// TwinCAT 3 PLC project PLC
// ProgramVersion: 3.1.4023.0
// libraries:
//   Tc2_Standard, * (Beckhoff Automation GmbH)
//   Tc2_System, * (Beckhoff Automation GmbH)
//   Tc3_Module, * (Beckhoff Automation GmbH)
// project tree:
//   / PlcTask.TcTTO
//   POUs/ MAIN.TcPOU
//   DUTs/IO/PdoEntries/ Status_B0753356.TcDUT, Status_F2CE6D91.TcDUT
//   DUTs/IO/PDOs/ InfoData_6F19DB2B.TcDUT, Channel_830843C1.TcDUT, WcState_9091E0EB.TcDUT, Channel_42CA91F7.TcDUT, WcState_0B2B16F9.TcDUT, AI_Standard_Channel_A8DF64E3.TcDUT, InfoData_32EB74EA.TcDUT, RTD_RTDInputs_Channel_A8DF64E3.TcDUT, AI_Standard_Channel_4A394481.TcDUT, TC_TCInputs_Channel_A8DF64E3.TcDUT, InfoData_E68C61CD.TcDUT, InfoData_2A97D6CF.TcDUT, Inputs_25A0042B.TcDUT, Outputs_2397A10E.TcDUT
//   DUTs/IO/Boxes/ EK1100_1FC0878B.TcDUT, EK1122_1FC0878B.TcDUT, EQ1008_78E8D3DD.TcDUT, EQ1809_32157CFD.TcDUT, EQ2008_E2806B95.TcDUT, EQ2339_4CF33DED.TcDUT, EQ2809_2B6483BD.TcDUT, EQ3174_DCC78662.TcDUT, EQ3204_6CD7E119.TcDUT, EQ3204_AB25C3AC.TcDUT, EQ3314_1CEB931C.TcDUT, EQ3314_E65CDB1C.TcDUT
//   DUTs/IO/Devices/ SyncUnitTask_2D604ED5.TcDUT, SyncUnitTasks_6FEB8257.TcDUT, SyncUnits_99E584AF.TcDUT
//   DUTs/IO/Topology/ Beckhoff_EQ1xxxEK1122_E78E0C94.TcDUT, Beckhoff_EQ1xxx_F67C323D.TcDUT, Beckhoff_EQ2xxxEK1122_214B8BB9.TcDUT, Beckhoff_EQ2xxx_A19B669C.TcDUT, Beckhoff_EQ3xxxEK1122_A1C56A21.TcDUT, Beckhoff_EQ3xxx_A920B096.TcDUT, EtherCAT_Master_EQxxxx_806C2CF0.TcDUT
//   DUTs/IO/Base/ EtcSlaveBase_82538BE2.TcDUT, EtcSlaveBase_82538BE2.TcDUT, EtcSlaveBase_82538BE2.TcDUT, EtcSlaveTerminalBase_947E5A46.TcDUT, EtcSlaveBoxBase_77A0E4A7.TcDUT, EtcSlaveEndTerminalBase_866C7F0C.TcDUT, InputBase_8311D824.TcDUT, OutputBase_10CEE7DE.TcDUT, EtcMasterBase_62654B43.TcDUT
//   GVLs/ GVL_iXlinker.TcGVL
// real-time tasks:
//   TASK PlcTask: cycle T#10ms, priority 20, ADS port 350
// I/O:
//   DEVICE EtherCAT_Master_EQxxxx, AmsNetId 172.20.30.238.15.1
//     Beckhoff EQ1xxx [EK1100 EtherCAT Coupler (2A E-Bus)]
//       Beckhoff EQ1xxxEK1122 [EK1122 2 port EtherCAT junction]
//         Beckhoff EQ1xxxsub EK1100 [EK1100 EtherCAT Coupler (2A E-Bus)]
//         A_0001(EQ1008-0002-0016) [EQ1008-0002 8 Ch. Dig. Input 24V, 3ms, M12]
//         A_0002(EQ1008-0002-0017) [EQ1008-0002 8 Ch. Dig. Input 24V, 3ms, M12]
//         A_0003(EQ1008-0002-0018) [EQ1008-0002 8 Ch. Dig. Input 24V, 3ms, M12]
//         A_0004(EQ1809-0022-0016) [EQ1809-0022 16 Ch. Dig. Input 24V, 3ms, M12]
//         A_0005(EQ1809-0022-0018) [EQ1809-0022 16 Ch. Dig. Input 24V, 3ms, M12]
//     Beckhoff EQ2xxx [EK1100 EtherCAT Coupler (2A E-Bus)]
//       Beckhoff EQ2xxxEK1122 [EK1122 2 port EtherCAT junction]
//         Beckhoff EQ2xxxsub EK1100 [EK1100 EtherCAT Coupler (2A E-Bus)]
//         A_0001(EQ2008-0002-0016) [EQ2008-0002 8 Ch. Dig. Output 24V, 0,5A, M12]
//         A_0002(EQ2008-0002-0017) [EQ2008-0002 8 Ch. Dig. Output 24V, 0,5A, M12]
//         A_0003(EQ2008-0002-0018) [EQ2008-0002 8 Ch. Dig. Output 24V, 0,5A, M12]
//         A_0004(EQ2008-0002-0019) [EQ2008-0002 8 Ch. Dig. Output 24V, 0,5A, M12]
//         A_0005(EQ2339-0022-0016) [EQ2339-0022 16 Ch. Dig. Input/Output 24V, 0,5A, M12]
//         A_0006(EQ2339-0022-0017) [EQ2339-0022 16 Ch. Dig. Input/Output 24V, 0,5A, M12]
//         A_0007(EQ2339-0022-0018) [EQ2339-0022 16 Ch. Dig. Input/Output 24V, 0,5A, M12]
//         A_0008(EQ2339-0022-0019) [EQ2339-0022 16 Ch. Dig. Input/Output 24V, 0,5A, M12]
//         A_0009(EQ2809-0022-0016) [EQ2809-0022 16 Ch. Dig. Output 24V, 0,5A, M12]
//         A_0010(EQ2809-0022-0017) [EQ2809-0022 16 Ch. Dig. Output 24V, 0,5A, M12]
//         A_0011(EQ2809-0022-0018) [EQ2809-0022 16 Ch. Dig. Output 24V, 0,5A, M12]
//     Beckhoff EQ3xxx [EK1100 EtherCAT Coupler (2A E-Bus)]
//       Beckhoff EQ3xxxEK1122 [EK1122 2 port EtherCAT junction]
//         Beckhoff EQ3xxxsub EK1100 [EK1100 EtherCAT Coupler (2A E-Bus)]
//         A_0001(EQ3174-0002-0016) [EQ3174-0002 4Ch. Ana. Input +/-10V, 0-10V, 0/4-20mA configurable]
//         A_0002(EQ3174-0002-0017) [EQ3174-0002 4Ch. Ana. Input +/-10V, 0-10V, 0/4-20mA configurable]
//         A_0003(EQ3174-0002-0021) [EQ3174-0002 4Ch. Ana. Input +/-10V, 0-10V, 0/4-20mA configurable]
//         A_0004(EQ3174-0002-0022) [EQ3174-0002 4Ch. Ana. Input +/-10V, 0-10V, 0/4-20mA configurable]
//         A_0005(EQ3174-0002-0023) [EQ3174-0002 4Ch. Ana. Input +/-10V, 0-10V, 0/4-20mA configurable]
//         A_0006(EQ3204-0002-0016) [EQ3204-0002 4Ch. Ana. Input PT100 (RTD)]
//         A_0007(EQ3204-0002-0017) [EQ3204-0002 4Ch. Ana. Input PT100 (RTD)]
//         A_0008(EQ3204-0002-0020) [EQ3204-0002 4Ch. Ana. Input PT100 (RTD)]
//         A_0009(EQ3204-0002-0021) [EQ3204-0002 4Ch. Ana. Input PT100 (RTD)]
//         A_0010(EQ3204-0002-0022) [EQ3204-0002 4Ch. Ana. Input PT100 (RTD)]
//         A_0011(EQ3314-0002-0016) [EQ3314-0002 4Ch. Ana. Input Thermocouple (TC)]
//         A_0012(EQ3314-0002-0017) [EQ3314-0002 4Ch. Ana. Input Thermocouple (TC)]
//         A_0013(EQ3314-0002-0021) [EQ3314-0002 4Ch. Ana. Input Thermocouple (TC)]
//         A_0014(EQ3314-0002-0022) [EQ3314-0002 4Ch. Ana. Input Thermocouple (TC)]
// variable links:
//   PLC/PLC Instance <-> EtherCAT Master EQxxxx/Beckhoff EQ1xxx
//     PlcTask Inputs/GVL_iXlinker.EtherCAT_Master_EQxxxx.Beckhoff_EQ1xxx.InfoData.State <-> InfoData/State
//   PLC/PLC Instance <-> EtherCAT Master EQxxxx/Beckhoff EQ1xxx/Beckhoff EQ1xxxEK1122
//     PlcTask Inputs/GVL_iXlinker.EtherCAT_Master_EQxxxx.Beckhoff_EQ1xxx.Beckhoff_EQ1xxxEK1122.InfoData.State <-> InfoData/State
//   PLC/PLC Instance <-> EtherCAT Master EQxxxx/Beckhoff EQ1xxx/Beckhoff EQ1xxxEK1122/Beckhoff EQ1xxxsub EK1100
//     PlcTask Inputs/GVL_iXlinker.EtherCAT_Master_EQxxxx.Beckhoff_EQ1xxx.Beckhoff_EQ1xxxEK1122.Beckhoff_EQ1xxxsub_EK1100.InfoData.State <-> InfoData/State
//   PLC/PLC Instance <-> EtherCAT Master EQxxxx/Beckhoff EQ1xxx/Beckhoff EQ1xxxEK1122/A_0001(EQ1008-0002-0016)
//     PlcTask Inputs/GVL_iXlinker.EtherCAT_Master_EQxxxx.Beckhoff_EQ1xxx.Beckhoff_EQ1xxxEK1122.A_0001_EQ1008_0002_0016.Channel_1.Input <-> Channel 1/Input
//     PlcTask Inputs/GVL_iXlinker.EtherCAT_Master_EQxxxx.Beckhoff_EQ1xxx.Beckhoff_EQ1xxxEK1122.A_0001_EQ1008_0002_0016.Channel_2.Input <-> Channel 2/Input
//     PlcTask Inputs/GVL_iXlinker.EtherCAT_Master_EQxxxx.Beckhoff_EQ1xxx.Beckhoff_EQ1xxxEK1122.A_0001_EQ1008_0002_0016.Channel_3.Input <-> Channel 3/Input
//     PlcTask Inputs/GVL_iXlinker.EtherCAT_Master_EQxxxx.Beckhoff_EQ1xxx.Beckhoff_EQ1xxxEK1122.A_0001_EQ1008_0002_0016.Channel_4.Input <-> Channel 4/Input
//     PlcTask Inputs/GVL_iXlinker.EtherCAT_Master_EQxxxx.Beckhoff_EQ1xxx.Beckhoff_EQ1xxxEK1122.A_0001_EQ1008_0002_0016.Channel_5.Input <-> Channel 5/Input
//     PlcTask Inputs/GVL_iXlinker.EtherCAT_Master_EQxxxx.Beckhoff_EQ1xxx.Beckhoff_EQ1xxxEK1122.A_0001_EQ1008_0002_0016.Channel_6.Input <-> Channel 6/Input
//     PlcTask Inputs/GVL_iXlinker.EtherCAT_Master_EQxxxx.Beckhoff_EQ1xxx.Beckhoff_EQ1xxxEK1122.A_0001_EQ1008_0002_0016.Channel_7.Input <-> Channel 7/Input
//     PlcTask Inputs/GVL_iXlinker.EtherCAT_Master_EQxxxx.Beckhoff_EQ1xxx.Beckhoff_EQ1xxxEK1122.A_0001_EQ1008_0002_0016.Channel_8.Input <-> Channel 8/Input
//     PlcTask Inputs/GVL_iXlinker.EtherCAT_Master_EQxxxx.Beckhoff_EQ1xxx.Beckhoff_EQ1xxxEK1122.A_0001_EQ1008_0002_0016.WcState.WcState <-> WcState/WcState
//     PlcTask Inputs/GVL_iXlinker.EtherCAT_Master_EQxxxx.Beckhoff_EQ1xxx.Beckhoff_EQ1xxxEK1122.A_0001_EQ1008_0002_0016.WcState.InputToggle <-> WcState/InputToggle
//     PlcTask Inputs/GVL_iXlinker.EtherCAT_Master_EQxxxx.Beckhoff_EQ1xxx.Beckhoff_EQ1xxxEK1122.A_0001_EQ1008_0002_0016.InfoData.State <-> InfoData/State
//   PLC/PLC Instance <-> EtherCAT Master EQxxxx/Beckhoff EQ1xxx/Beckhoff EQ1xxxEK1122/A_0002(EQ1008-0002-0017)
//     PlcTask Inputs/GVL_iXlinker.EtherCAT_Master_EQxxxx.Beckhoff_EQ1xxx.Beckhoff_EQ1xxxEK1122.A_0002_EQ1008_0002_0017.Channel_1.Input <-> Channel 1/Input
//     PlcTask Inputs/GVL_iXlinker.EtherCAT_Master_EQxxxx.Beckhoff_EQ1xxx.Beckhoff_EQ1xxxEK1122.A_0002_EQ1008_0002_0017.Channel_2.Input <-> Channel 2/Input
//     PlcTask Inputs/GVL_iXlinker.EtherCAT_Master_EQxxxx.Beckhoff_EQ1xxx.Beckhoff_EQ1xxxEK1122.A_0002_EQ1008_0002_0017.Channel_3.Input <-> Channel 3/Input
//     PlcTask Inputs/GVL_iXlinker.EtherCAT_Master_EQxxxx.Beckhoff_EQ1xxx.Beckhoff_EQ1xxxEK1122.A_0002_EQ1008_0002_0017.Channel_4.Input <-> Channel 4/Input
//     PlcTask Inputs/GVL_iXlinker.EtherCAT_Master_EQxxxx.Beckhoff_EQ1xxx.Beckhoff_EQ1xxxEK1122.A_0002_EQ1008_0002_0017.Channel_5.Input <-> Channel 5/Input
//     PlcTask Inputs/GVL_iXlinker.EtherCAT_Master_EQxxxx.Beckhoff_EQ1xxx.Beckhoff_EQ1xxxEK1122.A_0002_EQ1008_0002_0017.Channel_6.Input <-> Channel 6/Input
//     PlcTask Inputs/GVL_iXlinker.EtherCAT_Master_EQxxxx.Beckhoff_EQ1xxx.Beckhoff_EQ1xxxEK1122.A_0002_EQ1008_0002_0017.Channel_7.Input <-> Channel 7/Input
//     PlcTask Inputs/GVL_iXlinker.EtherCAT_Master_EQxxxx.Beckhoff_EQ1xxx.Beckhoff_EQ1xxxEK1122.A_0002_EQ1008_0002_0017.Channel_8.Input <-> Channel 8/Input
//     PlcTask Inputs/GVL_iXlinker.EtherCAT_Master_EQxxxx.Beckhoff_EQ1xxx.Beckhoff_EQ1xxxEK1122.A_0002_EQ1008_0002_0017.WcState.WcState <-> WcState/WcState
//     PlcTask Inputs/GVL_iXlinker.EtherCAT_Master_EQxxxx.Beckhoff_EQ1xxx.Beckhoff_EQ1xxxEK1122.A_0002_EQ1008_0002_0017.WcState.InputToggle <-> WcState/InputToggle
//     PlcTask Inputs/GVL_iXlinker.EtherCAT_Master_EQxxxx.Beckhoff_EQ1xxx.Beckhoff_EQ1xxxEK1122.A_0002_EQ1008_0002_0017.InfoData.State <-> InfoData/State
//   PLC/PLC Instance <-> EtherCAT Master EQxxxx/Beckhoff EQ1xxx/Beckhoff EQ1xxxEK1122/A_0003(EQ1008-0002-0018)
//     PlcTask Inputs/GVL_iXlinker.EtherCAT_Master_EQxxxx.Beckhoff_EQ1xxx.Beckhoff_EQ1xxxEK1122.A_0003_EQ1008_0002_0018.Channel_1.Input <-> Channel 1/Input
//     PlcTask Inputs/GVL_iXlinker.EtherCAT_Master_EQxxxx.Beckhoff_EQ1xxx.Beckhoff_EQ1xxxEK1122.A_0003_EQ1008_0002_0018.Channel_2.Input <-> Channel 2/Input
//     PlcTask Inputs/GVL_iXlinker.EtherCAT_Master_EQxxxx.Beckhoff_EQ1xxx.Beckhoff_EQ1xxxEK1122.A_0003_EQ1008_0002_0018.Channel_3.Input <-> Channel 3/Input
//     PlcTask Inputs/GVL_iXlinker.EtherCAT_Master_EQxxxx.Beckhoff_EQ1xxx.Beckhoff_EQ1xxxEK1122.A_0003_EQ1008_0002_0018.Channel_4.Input <-> Channel 4/Input
//     PlcTask Inputs/GVL_iXlinker.EtherCAT_Master_EQxxxx.Beckhoff_EQ1xxx.Beckhoff_EQ1xxxEK1122.A_0003_EQ1008_0002_0018.Channel_5.Input <-> Channel 5/Input
//     PlcTask Inputs/GVL_iXlinker.EtherCAT_Master_EQxxxx.Beckhoff_EQ1xxx.Beckhoff_EQ1xxxEK1122.A_0003_EQ1008_0002_0018.Channel_6.Input <-> Channel 6/Input
//     PlcTask Inputs/GVL_iXlinker.EtherCAT_Master_EQxxxx.Beckhoff_EQ1xxx.Beckhoff_EQ1xxxEK1122.A_0003_EQ1008_0002_0018.Channel_7.Input <-> Channel 7/Input
//     PlcTask Inputs/GVL_iXlinker.EtherCAT_Master_EQxxxx.Beckhoff_EQ1xxx.Beckhoff_EQ1xxxEK1122.A_0003_EQ1008_0002_0018.Channel_8.Input <-> Channel 8/Input
//     PlcTask Inputs/GVL_iXlinker.EtherCAT_Master_EQxxxx.Beckhoff_EQ1xxx.Beckhoff_EQ1xxxEK1122.A_0003_EQ1008_0002_0018.WcState.WcState <-> WcState/WcState
//     PlcTask Inputs/GVL_iXlinker.EtherCAT_Master_EQxxxx.Beckhoff_EQ1xxx.Beckhoff_EQ1xxxEK1122.A_0003_EQ1008_0002_0018.WcState.InputToggle <-> WcState/InputToggle
//     PlcTask Inputs/GVL_iXlinker.EtherCAT_Master_EQxxxx.Beckhoff_EQ1xxx.Beckhoff_EQ1xxxEK1122.A_0003_EQ1008_0002_0018.InfoData.State <-> InfoData/State
//   PLC/PLC Instance <-> EtherCAT Master EQxxxx/Beckhoff EQ1xxx/Beckhoff EQ1xxxEK1122/A_0004(EQ1809-0022-0016)
//     PlcTask Inputs/GVL_iXlinker.EtherCAT_Master_EQxxxx.Beckhoff_EQ1xxx.Beckhoff_EQ1xxxEK1122.A_0004_EQ1809_0022_0016.Channel_1.Input <-> Channel 1/Input
//     PlcTask Inputs/GVL_iXlinker.EtherCAT_Master_EQxxxx.Beckhoff_EQ1xxx.Beckhoff_EQ1xxxEK1122.A_0004_EQ1809_0022_0016.Channel_2.Input <-> Channel 2/Input
//     PlcTask Inputs/GVL_iXlinker.EtherCAT_Master_EQxxxx.Beckhoff_EQ1xxx.Beckhoff_EQ1xxxEK1122.A_0004_EQ1809_0022_0016.Channel_3.Input <-> Channel 3/Input
//     PlcTask Inputs/GVL_iXlinker.EtherCAT_Master_EQxxxx.Beckhoff_EQ1xxx.Beckhoff_EQ1xxxEK1122.A_0004_EQ1809_0022_0016.Channel_4.Input <-> Channel 4/Input
//     PlcTask Inputs/GVL_iXlinker.EtherCAT_Master_EQxxxx.Beckhoff_EQ1xxx.Beckhoff_EQ1xxxEK1122.A_0004_EQ1809_0022_0016.Channel_5.Input <-> Channel 5/Input
//     PlcTask Inputs/GVL_iXlinker.EtherCAT_Master_EQxxxx.Beckhoff_EQ1xxx.Beckhoff_EQ1xxxEK1122.A_0004_EQ1809_0022_0016.Channel_6.Input <-> Channel 6/Input
//     PlcTask Inputs/GVL_iXlinker.EtherCAT_Master_EQxxxx.Beckhoff_EQ1xxx.Beckhoff_EQ1xxxEK1122.A_0004_EQ1809_0022_0016.Channel_7.Input <-> Channel 7/Input
//     PlcTask Inputs/GVL_iXlinker.EtherCAT_Master_EQxxxx.Beckhoff_EQ1xxx.Beckhoff_EQ1xxxEK1122.A_0004_EQ1809_0022_0016.Channel_8.Input <-> Channel 8/Input
//     PlcTask Inputs/GVL_iXlinker.EtherCAT_Master_EQxxxx.Beckhoff_EQ1xxx.Beckhoff_EQ1xxxEK1122.A_0004_EQ1809_0022_0016.Channel_9.Input <-> Channel 9/Input
//     PlcTask Inputs/GVL_iXlinker.EtherCAT_Master_EQxxxx.Beckhoff_EQ1xxx.Beckhoff_EQ1xxxEK1122.A_0004_EQ1809_0022_0016.Channel_10.Input <-> Channel 10/Input
//     PlcTask Inputs/GVL_iXlinker.EtherCAT_Master_EQxxxx.Beckhoff_EQ1xxx.Beckhoff_EQ1xxxEK1122.A_0004_EQ1809_0022_0016.Channel_11.Input <-> Channel 11/Input
//     PlcTask Inputs/GVL_iXlinker.EtherCAT_Master_EQxxxx.Beckhoff_EQ1xxx.Beckhoff_EQ1xxxEK1122.A_0004_EQ1809_0022_0016.Channel_12.Input <-> Channel 12/Input
//     PlcTask Inputs/GVL_iXlinker.EtherCAT_Master_EQxxxx.Beckhoff_EQ1xxx.Beckhoff_EQ1xxxEK1122.A_0004_EQ1809_0022_0016.Channel_13.Input <-> Channel 13/Input
//     PlcTask Inputs/GVL_iXlinker.EtherCAT_Master_EQxxxx.Beckhoff_EQ1xxx.Beckhoff_EQ1xxxEK1122.A_0004_EQ1809_0022_0016.Channel_14.Input <-> Channel 14/Input
//     PlcTask Inputs/GVL_iXlinker.EtherCAT_Master_EQxxxx.Beckhoff_EQ1xxx.Beckhoff_EQ1xxxEK1122.A_0004_EQ1809_0022_0016.Channel_15.Input <-> Channel 15/Input
//     PlcTask Inputs/GVL_iXlinker.EtherCAT_Master_EQxxxx.Beckhoff_EQ1xxx.Beckhoff_EQ1xxxEK1122.A_0004_EQ1809_0022_0016.Channel_16.Input <-> Channel 16/Input
//     PlcTask Inputs/GVL_iXlinker.EtherCAT_Master_EQxxxx.Beckhoff_EQ1xxx.Beckhoff_EQ1xxxEK1122.A_0004_EQ1809_0022_0016.WcState.WcState <-> WcState/WcState
//     PlcTask Inputs/GVL_iXlinker.EtherCAT_Master_EQxxxx.Beckhoff_EQ1xxx.Beckhoff_EQ1xxxEK1122.A_0004_EQ1809_0022_0016.WcState.InputToggle <-> WcState/InputToggle
//     PlcTask Inputs/GVL_iXlinker.EtherCAT_Master_EQxxxx.Beckhoff_EQ1xxx.Beckhoff_EQ1xxxEK1122.A_0004_EQ1809_0022_0016.InfoData.State <-> InfoData/State
//   PLC/PLC Instance <-> EtherCAT Master EQxxxx/Beckhoff EQ1xxx/Beckhoff EQ1xxxEK1122/A_0005(EQ1809-0022-0018)
//     PlcTask Inputs/GVL_iXlinker.EtherCAT_Master_EQxxxx.Beckhoff_EQ1xxx.Beckhoff_EQ1xxxEK1122.A_0005_EQ1809_0022_0018.Channel_1.Input <-> Channel 1/Input
//     PlcTask Inputs/GVL_iXlinker.EtherCAT_Master_EQxxxx.Beckhoff_EQ1xxx.Beckhoff_EQ1xxxEK1122.A_0005_EQ1809_0022_0018.Channel_2.Input <-> Channel 2/Input
//     PlcTask Inputs/GVL_iXlinker.EtherCAT_Master_EQxxxx.Beckhoff_EQ1xxx.Beckhoff_EQ1xxxEK1122.A_0005_EQ1809_0022_0018.Channel_3.Input <-> Channel 3/Input
//     PlcTask Inputs/GVL_iXlinker.EtherCAT_Master_EQxxxx.Beckhoff_EQ1xxx.Beckhoff_EQ1xxxEK1122.A_0005_EQ1809_0022_0018.Channel_4.Input <-> Channel 4/Input
//     PlcTask Inputs/GVL_iXlinker.EtherCAT_Master_EQxxxx.Beckhoff_EQ1xxx.Beckhoff_EQ1xxxEK1122.A_0005_EQ1809_0022_0018.Channel_5.Input <-> Channel 5/Input
//     PlcTask Inputs/GVL_iXlinker.EtherCAT_Master_EQxxxx.Beckhoff_EQ1xxx.Beckhoff_EQ1xxxEK1122.A_0005_EQ1809_0022_0018.Channel_6.Input <-> Channel 6/Input
//     PlcTask Inputs/GVL_iXlinker.EtherCAT_Master_EQxxxx.Beckhoff_EQ1xxx.Beckhoff_EQ1xxxEK1122.A_0005_EQ1809_0022_0018.Channel_7.Input <-> Channel 7/Input
//     PlcTask Inputs/GVL_iXlinker.EtherCAT_Master_EQxxxx.Beckhoff_EQ1xxx.Beckhoff_EQ1xxxEK1122.A_0005_EQ1809_0022_0018.Channel_8.Input <-> Channel 8/Input
//     PlcTask Inputs/GVL_iXlinker.EtherCAT_Master_EQxxxx.Beckhoff_EQ1xxx.Beckhoff_EQ1xxxEK1122.A_0005_EQ1809_0022_0018.Channel_9.Input <-> Channel 9/Input
//     PlcTask Inputs/GVL_iXlinker.EtherCAT_Master_EQxxxx.Beckhoff_EQ1xxx.Beckhoff_EQ1xxxEK1122.A_0005_EQ1809_0022_0018.Channel_10.Input <-> Channel 10/Input
//     PlcTask Inputs/GVL_iXlinker.EtherCAT_Master_EQxxxx.Beckhoff_EQ1xxx.Beckhoff_EQ1xxxEK1122.A_0005_EQ1809_0022_0018.Channel_11.Input <-> Channel 11/Input
//     PlcTask Inputs/GVL_iXlinker.EtherCAT_Master_EQxxxx.Beckhoff_EQ1xxx.Beckhoff_EQ1xxxEK1122.A_0005_EQ1809_0022_0018.Channel_12.Input <-> Channel 12/Input
//     PlcTask Inputs/GVL_iXlinker.EtherCAT_Master_EQxxxx.Beckhoff_EQ1xxx.Beckhoff_EQ1xxxEK1122.A_0005_EQ1809_0022_0018.Channel_13.Input <-> Channel 13/Input
//     PlcTask Inputs/GVL_iXlinker.EtherCAT_Master_EQxxxx.Beckhoff_EQ1xxx.Beckhoff_EQ1xxxEK1122.A_0005_EQ1809_0022_0018.Channel_14.Input <-> Channel 14/Input
//     PlcTask Inputs/GVL_iXlinker.EtherCAT_Master_EQxxxx.Beckhoff_EQ1xxx.Beckhoff_EQ1xxxEK1122.A_0005_EQ1809_0022_0018.Channel_15.Input <-> Channel 15/Input
//     PlcTask Inputs/GVL_iXlinker.EtherCAT_Master_EQxxxx.Beckhoff_EQ1xxx.Beckhoff_EQ1xxxEK1122.A_0005_EQ1809_0022_0018.Channel_16.Input <-> Channel 16/Input
//     PlcTask Inputs/GVL_iXlinker.EtherCAT_Master_EQxxxx.Beckhoff_EQ1xxx.Beckhoff_EQ1xxxEK1122.A_0005_EQ1809_0022_0018.WcState.WcState <-> WcState/WcState
//     PlcTask Inputs/GVL_iXlinker.EtherCAT_Master_EQxxxx.Beckhoff_EQ1xxx.Beckhoff_EQ1xxxEK1122.A_0005_EQ1809_0022_0018.WcState.InputToggle <-> WcState/InputToggle
//     PlcTask Inputs/GVL_iXlinker.EtherCAT_Master_EQxxxx.Beckhoff_EQ1xxx.Beckhoff_EQ1xxxEK1122.A_0005_EQ1809_0022_0018.InfoData.State <-> InfoData/State
//   PLC/PLC Instance <-> EtherCAT Master EQxxxx/Beckhoff EQ2xxx
//     PlcTask Inputs/GVL_iXlinker.EtherCAT_Master_EQxxxx.Beckhoff_EQ2xxx.InfoData.State <-> InfoData/State
//   PLC/PLC Instance <-> EtherCAT Master EQxxxx/Beckhoff EQ2xxx/Beckhoff EQ2xxxEK1122
//     PlcTask Inputs/GVL_iXlinker.EtherCAT_Master_EQxxxx.Beckhoff_EQ2xxx.Beckhoff_EQ2xxxEK1122.InfoData.State <-> InfoData/State
//   PLC/PLC Instance <-> EtherCAT Master EQxxxx/Beckhoff EQ2xxx/Beckhoff EQ2xxxEK1122/Beckhoff EQ2xxxsub EK1100
//     PlcTask Inputs/GVL_iXlinker.EtherCAT_Master_EQxxxx.Beckhoff_EQ2xxx.Beckhoff_EQ2xxxEK1122.Beckhoff_EQ2xxxsub_EK1100.InfoData.State <-> InfoData/State
//   PLC/PLC Instance <-> EtherCAT Master EQxxxx/Beckhoff EQ2xxx/Beckhoff EQ2xxxEK1122/A_0001(EQ2008-0002-0016)
//     PlcTask Outputs/GVL_iXlinker.EtherCAT_Master_EQxxxx.Beckhoff_EQ2xxx.Beckhoff_EQ2xxxEK1122.A_0001_EQ2008_0002_0016.Channel_1.Output <-> Channel 1/Output
//     PlcTask Outputs/GVL_iXlinker.EtherCAT_Master_EQxxxx.Beckhoff_EQ2xxx.Beckhoff_EQ2xxxEK1122.A_0001_EQ2008_0002_0016.Channel_2.Output <-> Channel 2/Output
//     PlcTask Outputs/GVL_iXlinker.EtherCAT_Master_EQxxxx.Beckhoff_EQ2xxx.Beckhoff_EQ2xxxEK1122.A_0001_EQ2008_0002_0016.Channel_3.Output <-> Channel 3/Output
//     PlcTask Outputs/GVL_iXlinker.EtherCAT_Master_EQxxxx.Beckhoff_EQ2xxx.Beckhoff_EQ2xxxEK1122.A_0001_EQ2008_0002_0016.Channel_4.Output <-> Channel 4/Output
//     PlcTask Outputs/GVL_iXlinker.EtherCAT_Master_EQxxxx.Beckhoff_EQ2xxx.Beckhoff_EQ2xxxEK1122.A_0001_EQ2008_0002_0016.Channel_5.Output <-> Channel 5/Output
//     PlcTask Outputs/GVL_iXlinker.EtherCAT_Master_EQxxxx.Beckhoff_EQ2xxx.Beckhoff_EQ2xxxEK1122.A_0001_EQ2008_0002_0016.Channel_6.Output <-> Channel 6/Output
//     PlcTask Outputs/GVL_iXlinker.EtherCAT_Master_EQxxxx.Beckhoff_EQ2xxx.Beckhoff_EQ2xxxEK1122.A_0001_EQ2008_0002_0016.Channel_7.Output <-> Channel 7/Output
//     PlcTask Outputs/GVL_iXlinker.EtherCAT_Master_EQxxxx.Beckhoff_EQ2xxx.Beckhoff_EQ2xxxEK1122.A_0001_EQ2008_0002_0016.Channel_8.Output <-> Channel 8/Output
//     PlcTask Inputs/GVL_iXlinker.EtherCAT_Master_EQxxxx.Beckhoff_EQ2xxx.Beckhoff_EQ2xxxEK1122.A_0001_EQ2008_0002_0016.WcState.WcState <-> WcState/WcState
//     PlcTask Inputs/GVL_iXlinker.EtherCAT_Master_EQxxxx.Beckhoff_EQ2xxx.Beckhoff_EQ2xxxEK1122.A_0001_EQ2008_0002_0016.InfoData.State <-> InfoData/State
//   PLC/PLC Instance <-> EtherCAT Master EQxxxx/Beckhoff EQ2xxx/Beckhoff EQ2xxxEK1122/A_0002(EQ2008-0002-0017)
//     PlcTask Outputs/GVL_iXlinker.EtherCAT_Master_EQxxxx.Beckhoff_EQ2xxx.Beckhoff_EQ2xxxEK1122.A_0002_EQ2008_0002_0017.Channel_1.Output <-> Channel 1/Output
//     PlcTask Outputs/GVL_iXlinker.EtherCAT_Master_EQxxxx.Beckhoff_EQ2xxx.Beckhoff_EQ2xxxEK1122.A_0002_EQ2008_0002_0017.Channel_2.Output <-> Channel 2/Output
//     PlcTask Outputs/GVL_iXlinker.EtherCAT_Master_EQxxxx.Beckhoff_EQ2xxx.Beckhoff_EQ2xxxEK1122.A_0002_EQ2008_0002_0017.Channel_3.Output <-> Channel 3/Output
//     PlcTask Outputs/GVL_iXlinker.EtherCAT_Master_EQxxxx.Beckhoff_EQ2xxx.Beckhoff_EQ2xxxEK1122.A_0002_EQ2008_0002_0017.Channel_4.Output <-> Channel 4/Output
//     PlcTask Outputs/GVL_iXlinker.EtherCAT_Master_EQxxxx.Beckhoff_EQ2xxx.Beckhoff_EQ2xxxEK1122.A_0002_EQ2008_0002_0017.Channel_5.Output <-> Channel 5/Output
//     PlcTask Outputs/GVL_iXlinker.EtherCAT_Master_EQxxxx.Beckhoff_EQ2xxx.Beckhoff_EQ2xxxEK1122.A_0002_EQ2008_0002_0017.Channel_6.Output <-> Channel 6/Output
//     PlcTask Outputs/GVL_iXlinker.EtherCAT_Master_EQxxxx.Beckhoff_EQ2xxx.Beckhoff_EQ2xxxEK1122.A_0002_EQ2008_0002_0017.Channel_7.Output <-> Channel 7/Output
//     PlcTask Outputs/GVL_iXlinker.EtherCAT_Master_EQxxxx.Beckhoff_EQ2xxx.Beckhoff_EQ2xxxEK1122.A_0002_EQ2008_0002_0017.Channel_8.Output <-> Channel 8/Output
//     PlcTask Inputs/GVL_iXlinker.EtherCAT_Master_EQxxxx.Beckhoff_EQ2xxx.Beckhoff_EQ2xxxEK1122.A_0002_EQ2008_0002_0017.WcState.WcState <-> WcState/WcState
//     PlcTask Inputs/GVL_iXlinker.EtherCAT_Master_EQxxxx.Beckhoff_EQ2xxx.Beckhoff_EQ2xxxEK1122.A_0002_EQ2008_0002_0017.InfoData.State <-> InfoData/State
//   PLC/PLC Instance <-> EtherCAT Master EQxxxx/Beckhoff EQ2xxx/Beckhoff EQ2xxxEK1122/A_0003(EQ2008-0002-0018)
//     PlcTask Outputs/GVL_iXlinker.EtherCAT_Master_EQxxxx.Beckhoff_EQ2xxx.Beckhoff_EQ2xxxEK1122.A_0003_EQ2008_0002_0018.Channel_1.Output <-> Channel 1/Output
//     PlcTask Outputs/GVL_iXlinker.EtherCAT_Master_EQxxxx.Beckhoff_EQ2xxx.Beckhoff_EQ2xxxEK1122.A_0003_EQ2008_0002_0018.Channel_2.Output <-> Channel 2/Output
//     PlcTask Outputs/GVL_iXlinker.EtherCAT_Master_EQxxxx.Beckhoff_EQ2xxx.Beckhoff_EQ2xxxEK1122.A_0003_EQ2008_0002_0018.Channel_3.Output <-> Channel 3/Output
//     PlcTask Outputs/GVL_iXlinker.EtherCAT_Master_EQxxxx.Beckhoff_EQ2xxx.Beckhoff_EQ2xxxEK1122.A_0003_EQ2008_0002_0018.Channel_4.Output <-> Channel 4/Output
//     PlcTask Outputs/GVL_iXlinker.EtherCAT_Master_EQxxxx.Beckhoff_EQ2xxx.Beckhoff_EQ2xxxEK1122.A_0003_EQ2008_0002_0018.Channel_5.Output <-> Channel 5/Output
//     PlcTask Outputs/GVL_iXlinker.EtherCAT_Master_EQxxxx.Beckhoff_EQ2xxx.Beckhoff_EQ2xxxEK1122.A_0003_EQ2008_0002_0018.Channel_6.Output <-> Channel 6/Output
//     PlcTask Outputs/GVL_iXlinker.EtherCAT_Master_EQxxxx.Beckhoff_EQ2xxx.Beckhoff_EQ2xxxEK1122.A_0003_EQ2008_0002_0018.Channel_7.Output <-> Channel 7/Output
//     PlcTask Outputs/GVL_iXlinker.EtherCAT_Master_EQxxxx.Beckhoff_EQ2xxx.Beckhoff_EQ2xxxEK1122.A_0003_EQ2008_0002_0018.Channel_8.Output <-> Channel 8/Output
//     PlcTask Inputs/GVL_iXlinker.EtherCAT_Master_EQxxxx.Beckhoff_EQ2xxx.Beckhoff_EQ2xxxEK1122.A_0003_EQ2008_0002_0018.WcState.WcState <-> WcState/WcState
//     PlcTask Inputs/GVL_iXlinker.EtherCAT_Master_EQxxxx.Beckhoff_EQ2xxx.Beckhoff_EQ2xxxEK1122.A_0003_EQ2008_0002_0018.InfoData.State <-> InfoData/State
//   PLC/PLC Instance <-> EtherCAT Master EQxxxx/Beckhoff EQ2xxx/Beckhoff EQ2xxxEK1122/A_0004(EQ2008-0002-0019)
//     PlcTask Outputs/GVL_iXlinker.EtherCAT_Master_EQxxxx.Beckhoff_EQ2xxx.Beckhoff_EQ2xxxEK1122.A_0004_EQ2008_0002_0019.Channel_1.Output <-> Channel 1/Output
//     PlcTask Outputs/GVL_iXlinker.EtherCAT_Master_EQxxxx.Beckhoff_EQ2xxx.Beckhoff_EQ2xxxEK1122.A_0004_EQ2008_0002_0019.Channel_2.Output <-> Channel 2/Output
//     PlcTask Outputs/GVL_iXlinker.EtherCAT_Master_EQxxxx.Beckhoff_EQ2xxx.Beckhoff_EQ2xxxEK1122.A_0004_EQ2008_0002_0019.Channel_3.Output <-> Channel 3/Output
//     PlcTask Outputs/GVL_iXlinker.EtherCAT_Master_EQxxxx.Beckhoff_EQ2xxx.Beckhoff_EQ2xxxEK1122.A_0004_EQ2008_0002_0019.Channel_4.Output <-> Channel 4/Output
//     PlcTask Outputs/GVL_iXlinker.EtherCAT_Master_EQxxxx.Beckhoff_EQ2xxx.Beckhoff_EQ2xxxEK1122.A_0004_EQ2008_0002_0019.Channel_5.Output <-> Channel 5/Output
//     PlcTask Outputs/GVL_iXlinker.EtherCAT_Master_EQxxxx.Beckhoff_EQ2xxx.Beckhoff_EQ2xxxEK1122.A_0004_EQ2008_0002_0019.Channel_6.Output <-> Channel 6/Output
//     PlcTask Outputs/GVL_iXlinker.EtherCAT_Master_EQxxxx.Beckhoff_EQ2xxx.Beckhoff_EQ2xxxEK1122.A_0004_EQ2008_0002_0019.Channel_7.Output <-> Channel 7/Output
//     PlcTask Outputs/GVL_iXlinker.EtherCAT_Master_EQxxxx.Beckhoff_EQ2xxx.Beckhoff_EQ2xxxEK1122.A_0004_EQ2008_0002_0019.Channel_8.Output <-> Channel 8/Output
//     PlcTask Inputs/GVL_iXlinker.EtherCAT_Master_EQxxxx.Beckhoff_EQ2xxx.Beckhoff_EQ2xxxEK1122.A_0004_EQ2008_0002_0019.WcState.WcState <-> WcState/WcState
//     PlcTask Inputs/GVL_iXlinker.EtherCAT_Master_EQxxxx.Beckhoff_EQ2xxx.Beckhoff_EQ2xxxEK1122.A_0004_EQ2008_0002_0019.InfoData.State <-> InfoData/State
//   PLC/PLC Instance <-> EtherCAT Master EQxxxx/Beckhoff EQ2xxx/Beckhoff EQ2xxxEK1122/A_0005(EQ2339-0022-0016)
//     PlcTask Inputs/GVL_iXlinker.EtherCAT_Master_EQxxxx.Beckhoff_EQ2xxx.Beckhoff_EQ2xxxEK1122.A_0005_EQ2339_0022_0016.Channel_1.Input <-> Channel 1/Input
//     PlcTask Inputs/GVL_iXlinker.EtherCAT_Master_EQxxxx.Beckhoff_EQ2xxx.Beckhoff_EQ2xxxEK1122.A_0005_EQ2339_0022_0016.Channel_2.Input <-> Channel 2/Input
//     PlcTask Inputs/GVL_iXlinker.EtherCAT_Master_EQxxxx.Beckhoff_EQ2xxx.Beckhoff_EQ2xxxEK1122.A_0005_EQ2339_0022_0016.Channel_3.Input <-> Channel 3/Input
//     PlcTask Inputs/GVL_iXlinker.EtherCAT_Master_EQxxxx.Beckhoff_EQ2xxx.Beckhoff_EQ2xxxEK1122.A_0005_EQ2339_0022_0016.Channel_4.Input <-> Channel 4/Input
//     PlcTask Inputs/GVL_iXlinker.EtherCAT_Master_EQxxxx.Beckhoff_EQ2xxx.Beckhoff_EQ2xxxEK1122.A_0005_EQ2339_0022_0016.Channel_5.Input <-> Channel 5/Input
//     PlcTask Inputs/GVL_iXlinker.EtherCAT_Master_EQxxxx.Beckhoff_EQ2xxx.Beckhoff_EQ2xxxEK1122.A_0005_EQ2339_0022_0016.Channel_6.Input <-> Channel 6/Input
//     PlcTask Inputs/GVL_iXlinker.EtherCAT_Master_EQxxxx.Beckhoff_EQ2xxx.Beckhoff_EQ2xxxEK1122.A_0005_EQ2339_0022_0016.Channel_7.Input <-> Channel 7/Input
//     PlcTask Inputs/GVL_iXlinker.EtherCAT_Master_EQxxxx.Beckhoff_EQ2xxx.Beckhoff_EQ2xxxEK1122.A_0005_EQ2339_0022_0016.Channel_8.Input <-> Channel 8/Input
//     PlcTask Inputs/GVL_iXlinker.EtherCAT_Master_EQxxxx.Beckhoff_EQ2xxx.Beckhoff_EQ2xxxEK1122.A_0005_EQ2339_0022_0016.Channel_9.Input <-> Channel 9/Input
//     PlcTask Inputs/GVL_iXlinker.EtherCAT_Master_EQxxxx.Beckhoff_EQ2xxx.Beckhoff_EQ2xxxEK1122.A_0005_EQ2339_0022_0016.Channel_10.Input <-> Channel 10/Input
//     PlcTask Inputs/GVL_iXlinker.EtherCAT_Master_EQxxxx.Beckhoff_EQ2xxx.Beckhoff_EQ2xxxEK1122.A_0005_EQ2339_0022_0016.Channel_11.Input <-> Channel 11/Input
//     PlcTask Inputs/GVL_iXlinker.EtherCAT_Master_EQxxxx.Beckhoff_EQ2xxx.Beckhoff_EQ2xxxEK1122.A_0005_EQ2339_0022_0016.Channel_12.Input <-> Channel 12/Input
//     PlcTask Inputs/GVL_iXlinker.EtherCAT_Master_EQxxxx.Beckhoff_EQ2xxx.Beckhoff_EQ2xxxEK1122.A_0005_EQ2339_0022_0016.Channel_13.Input <-> Channel 13/Input
//     PlcTask Inputs/GVL_iXlinker.EtherCAT_Master_EQxxxx.Beckhoff_EQ2xxx.Beckhoff_EQ2xxxEK1122.A_0005_EQ2339_0022_0016.Channel_14.Input <-> Channel 14/Input
//     PlcTask Inputs/GVL_iXlinker.EtherCAT_Master_EQxxxx.Beckhoff_EQ2xxx.Beckhoff_EQ2xxxEK1122.A_0005_EQ2339_0022_0016.Channel_15.Input <-> Channel 15/Input
//     PlcTask Inputs/GVL_iXlinker.EtherCAT_Master_EQxxxx.Beckhoff_EQ2xxx.Beckhoff_EQ2xxxEK1122.A_0005_EQ2339_0022_0016.Channel_16.Input <-> Channel 16/Input
//     PlcTask Outputs/GVL_iXlinker.EtherCAT_Master_EQxxxx.Beckhoff_EQ2xxx.Beckhoff_EQ2xxxEK1122.A_0005_EQ2339_0022_0016.Channel_17.Output <-> Channel 17/Output
//     PlcTask Outputs/GVL_iXlinker.EtherCAT_Master_EQxxxx.Beckhoff_EQ2xxx.Beckhoff_EQ2xxxEK1122.A_0005_EQ2339_0022_0016.Channel_18.Output <-> Channel 18/Output
//     PlcTask Outputs/GVL_iXlinker.EtherCAT_Master_EQxxxx.Beckhoff_EQ2xxx.Beckhoff_EQ2xxxEK1122.A_0005_EQ2339_0022_0016.Channel_19.Output <-> Channel 19/Output
//     PlcTask Outputs/GVL_iXlinker.EtherCAT_Master_EQxxxx.Beckhoff_EQ2xxx.Beckhoff_EQ2xxxEK1122.A_0005_EQ2339_0022_0016.Channel_20.Output <-> Channel 20/Output
//     PlcTask Outputs/GVL_iXlinker.EtherCAT_Master_EQxxxx.Beckhoff_EQ2xxx.Beckhoff_EQ2xxxEK1122.A_0005_EQ2339_0022_0016.Channel_21.Output <-> Channel 21/Output
//     PlcTask Outputs/GVL_iXlinker.EtherCAT_Master_EQxxxx.Beckhoff_EQ2xxx.Beckhoff_EQ2xxxEK1122.A_0005_EQ2339_0022_0016.Channel_22.Output <-> Channel 22/Output
//     PlcTask Outputs/GVL_iXlinker.EtherCAT_Master_EQxxxx.Beckhoff_EQ2xxx.Beckhoff_EQ2xxxEK1122.A_0005_EQ2339_0022_0016.Channel_23.Output <-> Channel 23/Output
//     PlcTask Outputs/GVL_iXlinker.EtherCAT_Master_EQxxxx.Beckhoff_EQ2xxx.Beckhoff_EQ2xxxEK1122.A_0005_EQ2339_0022_0016.Channel_24.Output <-> Channel 24/Output
//     PlcTask Outputs/GVL_iXlinker.EtherCAT_Master_EQxxxx.Beckhoff_EQ2xxx.Beckhoff_EQ2xxxEK1122.A_0005_EQ2339_0022_0016.Channel_25.Output <-> Channel 25/Output
//     PlcTask Outputs/GVL_iXlinker.EtherCAT_Master_EQxxxx.Beckhoff_EQ2xxx.Beckhoff_EQ2xxxEK1122.A_0005_EQ2339_0022_0016.Channel_26.Output <-> Channel 26/Output
//     PlcTask Outputs/GVL_iXlinker.EtherCAT_Master_EQxxxx.Beckhoff_EQ2xxx.Beckhoff_EQ2xxxEK1122.A_0005_EQ2339_0022_0016.Channel_27.Output <-> Channel 27/Output
//     PlcTask Outputs/GVL_iXlinker.EtherCAT_Master_EQxxxx.Beckhoff_EQ2xxx.Beckhoff_EQ2xxxEK1122.A_0005_EQ2339_0022_0016.Channel_28.Output <-> Channel 28/Output
//     PlcTask Outputs/GVL_iXlinker.EtherCAT_Master_EQxxxx.Beckhoff_EQ2xxx.Beckhoff_EQ2xxxEK1122.A_0005_EQ2339_0022_0016.Channel_29.Output <-> Channel 29/Output
//     PlcTask Outputs/GVL_iXlinker.EtherCAT_Master_EQxxxx.Beckhoff_EQ2xxx.Beckhoff_EQ2xxxEK1122.A_0005_EQ2339_0022_0016.Channel_30.Output <-> Channel 30/Output
//     PlcTask Outputs/GVL_iXlinker.EtherCAT_Master_EQxxxx.Beckhoff_EQ2xxx.Beckhoff_EQ2xxxEK1122.A_0005_EQ2339_0022_0016.Channel_31.Output <-> Channel 31/Output
//     PlcTask Outputs/GVL_iXlinker.EtherCAT_Master_EQxxxx.Beckhoff_EQ2xxx.Beckhoff_EQ2xxxEK1122.A_0005_EQ2339_0022_0016.Channel_32.Output <-> Channel 32/Output
//     PlcTask Inputs/GVL_iXlinker.EtherCAT_Master_EQxxxx.Beckhoff_EQ2xxx.Beckhoff_EQ2xxxEK1122.A_0005_EQ2339_0022_0016.WcState.WcState <-> WcState/WcState
//     PlcTask Inputs/GVL_iXlinker.EtherCAT_Master_EQxxxx.Beckhoff_EQ2xxx.Beckhoff_EQ2xxxEK1122.A_0005_EQ2339_0022_0016.WcState.InputToggle <-> WcState/InputToggle
//     PlcTask Inputs/GVL_iXlinker.EtherCAT_Master_EQxxxx.Beckhoff_EQ2xxx.Beckhoff_EQ2xxxEK1122.A_0005_EQ2339_0022_0016.InfoData.State <-> InfoData/State
//   PLC/PLC Instance <-> EtherCAT Master EQxxxx/Beckhoff EQ2xxx/Beckhoff EQ2xxxEK1122/A_0006(EQ2339-0022-0017)
//     PlcTask Inputs/GVL_iXlinker.EtherCAT_Master_EQxxxx.Beckhoff_EQ2xxx.Beckhoff_EQ2xxxEK1122.A_0006_EQ2339_0022_0017.Channel_1.Input <-> Channel 1/Input
//     PlcTask Inputs/GVL_iXlinker.EtherCAT_Master_EQxxxx.Beckhoff_EQ2xxx.Beckhoff_EQ2xxxEK1122.A_0006_EQ2339_0022_0017.Channel_2.Input <-> Channel 2/Input
//     PlcTask Inputs/GVL_iXlinker.EtherCAT_Master_EQxxxx.Beckhoff_EQ2xxx.Beckhoff_EQ2xxxEK1122.A_0006_EQ2339_0022_0017.Channel_3.Input <-> Channel 3/Input
//     PlcTask Inputs/GVL_iXlinker.EtherCAT_Master_EQxxxx.Beckhoff_EQ2xxx.Beckhoff_EQ2xxxEK1122.A_0006_EQ2339_0022_0017.Channel_4.Input <-> Channel 4/Input
//     PlcTask Inputs/GVL_iXlinker.EtherCAT_Master_EQxxxx.Beckhoff_EQ2xxx.Beckhoff_EQ2xxxEK1122.A_0006_EQ2339_0022_0017.Channel_5.Input <-> Channel 5/Input
//     PlcTask Inputs/GVL_iXlinker.EtherCAT_Master_EQxxxx.Beckhoff_EQ2xxx.Beckhoff_EQ2xxxEK1122.A_0006_EQ2339_0022_0017.Channel_6.Input <-> Channel 6/Input
//     PlcTask Inputs/GVL_iXlinker.EtherCAT_Master_EQxxxx.Beckhoff_EQ2xxx.Beckhoff_EQ2xxxEK1122.A_0006_EQ2339_0022_0017.Channel_7.Input <-> Channel 7/Input
//     PlcTask Inputs/GVL_iXlinker.EtherCAT_Master_EQxxxx.Beckhoff_EQ2xxx.Beckhoff_EQ2xxxEK1122.A_0006_EQ2339_0022_0017.Channel_8.Input <-> Channel 8/Input
//     PlcTask Inputs/GVL_iXlinker.EtherCAT_Master_EQxxxx.Beckhoff_EQ2xxx.Beckhoff_EQ2xxxEK1122.A_0006_EQ2339_0022_0017.Channel_9.Input <-> Channel 9/Input
//     PlcTask Inputs/GVL_iXlinker.EtherCAT_Master_EQxxxx.Beckhoff_EQ2xxx.Beckhoff_EQ2xxxEK1122.A_0006_EQ2339_0022_0017.Channel_10.Input <-> Channel 10/Input
//     PlcTask Inputs/GVL_iXlinker.EtherCAT_Master_EQxxxx.Beckhoff_EQ2xxx.Beckhoff_EQ2xxxEK1122.A_0006_EQ2339_0022_0017.Channel_11.Input <-> Channel 11/Input
//     PlcTask Inputs/GVL_iXlinker.EtherCAT_Master_EQxxxx.Beckhoff_EQ2xxx.Beckhoff_EQ2xxxEK1122.A_0006_EQ2339_0022_0017.Channel_12.Input <-> Channel 12/Input
//     PlcTask Inputs/GVL_iXlinker.EtherCAT_Master_EQxxxx.Beckhoff_EQ2xxx.Beckhoff_EQ2xxxEK1122.A_0006_EQ2339_0022_0017.Channel_13.Input <-> Channel 13/Input
//     PlcTask Inputs/GVL_iXlinker.EtherCAT_Master_EQxxxx.Beckhoff_EQ2xxx.Beckhoff_EQ2xxxEK1122.A_0006_EQ2339_0022_0017.Channel_14.Input <-> Channel 14/Input
//     PlcTask Inputs/GVL_iXlinker.EtherCAT_Master_EQxxxx.Beckhoff_EQ2xxx.Beckhoff_EQ2xxxEK1122.A_0006_EQ2339_0022_0017.Channel_15.Input <-> Channel 15/Input
//     PlcTask Inputs/GVL_iXlinker.EtherCAT_Master_EQxxxx.Beckhoff_EQ2xxx.Beckhoff_EQ2xxxEK1122.A_0006_EQ2339_0022_0017.Channel_16.Input <-> Channel 16/Input
//     PlcTask Outputs/GVL_iXlinker.EtherCAT_Master_EQxxxx.Beckhoff_EQ2xxx.Beckhoff_EQ2xxxEK1122.A_0006_EQ2339_0022_0017.Channel_17.Output <-> Channel 17/Output
//     PlcTask Outputs/GVL_iXlinker.EtherCAT_Master_EQxxxx.Beckhoff_EQ2xxx.Beckhoff_EQ2xxxEK1122.A_0006_EQ2339_0022_0017.Channel_18.Output <-> Channel 18/Output
//     PlcTask Outputs/GVL_iXlinker.EtherCAT_Master_EQxxxx.Beckhoff_EQ2xxx.Beckhoff_EQ2xxxEK1122.A_0006_EQ2339_0022_0017.Channel_19.Output <-> Channel 19/Output
//     PlcTask Outputs/GVL_iXlinker.EtherCAT_Master_EQxxxx.Beckhoff_EQ2xxx.Beckhoff_EQ2xxxEK1122.A_0006_EQ2339_0022_0017.Channel_20.Output <-> Channel 20/Output
//     PlcTask Outputs/GVL_iXlinker.EtherCAT_Master_EQxxxx.Beckhoff_EQ2xxx.Beckhoff_EQ2xxxEK1122.A_0006_EQ2339_0022_0017.Channel_21.Output <-> Channel 21/Output
//     PlcTask Outputs/GVL_iXlinker.EtherCAT_Master_EQxxxx.Beckhoff_EQ2xxx.Beckhoff_EQ2xxxEK1122.A_0006_EQ2339_0022_0017.Channel_22.Output <-> Channel 22/Output
//     PlcTask Outputs/GVL_iXlinker.EtherCAT_Master_EQxxxx.Beckhoff_EQ2xxx.Beckhoff_EQ2xxxEK1122.A_0006_EQ2339_0022_0017.Channel_23.Output <-> Channel 23/Output
//     PlcTask Outputs/GVL_iXlinker.EtherCAT_Master_EQxxxx.Beckhoff_EQ2xxx.Beckhoff_EQ2xxxEK1122.A_0006_EQ2339_0022_0017.Channel_24.Output <-> Channel 24/Output
//     PlcTask Outputs/GVL_iXlinker.EtherCAT_Master_EQxxxx.Beckhoff_EQ2xxx.Beckhoff_EQ2xxxEK1122.A_0006_EQ2339_0022_0017.Channel_25.Output <-> Channel 25/Output
//     PlcTask Outputs/GVL_iXlinker.EtherCAT_Master_EQxxxx.Beckhoff_EQ2xxx.Beckhoff_EQ2xxxEK1122.A_0006_EQ2339_0022_0017.Channel_26.Output <-> Channel 26/Output
//     PlcTask Outputs/GVL_iXlinker.EtherCAT_Master_EQxxxx.Beckhoff_EQ2xxx.Beckhoff_EQ2xxxEK1122.A_0006_EQ2339_0022_0017.Channel_27.Output <-> Channel 27/Output
//     PlcTask Outputs/GVL_iXlinker.EtherCAT_Master_EQxxxx.Beckhoff_EQ2xxx.Beckhoff_EQ2xxxEK1122.A_0006_EQ2339_0022_0017.Channel_28.Output <-> Channel 28/Output
//     PlcTask Outputs/GVL_iXlinker.EtherCAT_Master_EQxxxx.Beckhoff_EQ2xxx.Beckhoff_EQ2xxxEK1122.A_0006_EQ2339_0022_0017.Channel_29.Output <-> Channel 29/Output
//     PlcTask Outputs/GVL_iXlinker.EtherCAT_Master_EQxxxx.Beckhoff_EQ2xxx.Beckhoff_EQ2xxxEK1122.A_0006_EQ2339_0022_0017.Channel_30.Output <-> Channel 30/Output
//     PlcTask Outputs/GVL_iXlinker.EtherCAT_Master_EQxxxx.Beckhoff_EQ2xxx.Beckhoff_EQ2xxxEK1122.A_0006_EQ2339_0022_0017.Channel_31.Output <-> Channel 31/Output
//     PlcTask Outputs/GVL_iXlinker.EtherCAT_Master_EQxxxx.Beckhoff_EQ2xxx.Beckhoff_EQ2xxxEK1122.A_0006_EQ2339_0022_0017.Channel_32.Output <-> Channel 32/Output
//     PlcTask Inputs/GVL_iXlinker.EtherCAT_Master_EQxxxx.Beckhoff_EQ2xxx.Beckhoff_EQ2xxxEK1122.A_0006_EQ2339_0022_0017.WcState.WcState <-> WcState/WcState
//     PlcTask Inputs/GVL_iXlinker.EtherCAT_Master_EQxxxx.Beckhoff_EQ2xxx.Beckhoff_EQ2xxxEK1122.A_0006_EQ2339_0022_0017.WcState.InputToggle <-> WcState/InputToggle
//     PlcTask Inputs/GVL_iXlinker.EtherCAT_Master_EQxxxx.Beckhoff_EQ2xxx.Beckhoff_EQ2xxxEK1122.A_0006_EQ2339_0022_0017.InfoData.State <-> InfoData/State
//   PLC/PLC Instance <-> EtherCAT Master EQxxxx/Beckhoff EQ2xxx/Beckhoff EQ2xxxEK1122/A_0007(EQ2339-0022-0018)
//     PlcTask Inputs/GVL_iXlinker.EtherCAT_Master_EQxxxx.Beckhoff_EQ2xxx.Beckhoff_EQ2xxxEK1122.A_0007_EQ2339_0022_0018.Channel_1.Input <-> Channel 1/Input
//     PlcTask Inputs/GVL_iXlinker.EtherCAT_Master_EQxxxx.Beckhoff_EQ2xxx.Beckhoff_EQ2xxxEK1122.A_0007_EQ2339_0022_0018.Channel_2.Input <-> Channel 2/Input
//     PlcTask Inputs/GVL_iXlinker.EtherCAT_Master_EQxxxx.Beckhoff_EQ2xxx.Beckhoff_EQ2xxxEK1122.A_0007_EQ2339_0022_0018.Channel_3.Input <-> Channel 3/Input
//     PlcTask Inputs/GVL_iXlinker.EtherCAT_Master_EQxxxx.Beckhoff_EQ2xxx.Beckhoff_EQ2xxxEK1122.A_0007_EQ2339_0022_0018.Channel_4.Input <-> Channel 4/Input
//     PlcTask Inputs/GVL_iXlinker.EtherCAT_Master_EQxxxx.Beckhoff_EQ2xxx.Beckhoff_EQ2xxxEK1122.A_0007_EQ2339_0022_0018.Channel_5.Input <-> Channel 5/Input
//     PlcTask Inputs/GVL_iXlinker.EtherCAT_Master_EQxxxx.Beckhoff_EQ2xxx.Beckhoff_EQ2xxxEK1122.A_0007_EQ2339_0022_0018.Channel_6.Input <-> Channel 6/Input
//     PlcTask Inputs/GVL_iXlinker.EtherCAT_Master_EQxxxx.Beckhoff_EQ2xxx.Beckhoff_EQ2xxxEK1122.A_0007_EQ2339_0022_0018.Channel_7.Input <-> Channel 7/Input
//     PlcTask Inputs/GVL_iXlinker.EtherCAT_Master_EQxxxx.Beckhoff_EQ2xxx.Beckhoff_EQ2xxxEK1122.A_0007_EQ2339_0022_0018.Channel_8.Input <-> Channel 8/Input
//     PlcTask Inputs/GVL_iXlinker.EtherCAT_Master_EQxxxx.Beckhoff_EQ2xxx.Beckhoff_EQ2xxxEK1122.A_0007_EQ2339_0022_0018.Channel_9.Input <-> Channel 9/Input
//     PlcTask Inputs/GVL_iXlinker.EtherCAT_Master_EQxxxx.Beckhoff_EQ2xxx.Beckhoff_EQ2xxxEK1122.A_0007_EQ2339_0022_0018.Channel_10.Input <-> Channel 10/Input
//     PlcTask Inputs/GVL_iXlinker.EtherCAT_Master_EQxxxx.Beckhoff_EQ2xxx.Beckhoff_EQ2xxxEK1122.A_0007_EQ2339_0022_0018.Channel_11.Input <-> Channel 11/Input
//     PlcTask Inputs/GVL_iXlinker.EtherCAT_Master_EQxxxx.Beckhoff_EQ2xxx.Beckhoff_EQ2xxxEK1122.A_0007_EQ2339_0022_0018.Channel_12.Input <-> Channel 12/Input
//     PlcTask Inputs/GVL_iXlinker.EtherCAT_Master_EQxxxx.Beckhoff_EQ2xxx.Beckhoff_EQ2xxxEK1122.A_0007_EQ2339_0022_0018.Channel_13.Input <-> Channel 13/Input
//     PlcTask Inputs/GVL_iXlinker.EtherCAT_Master_EQxxxx.Beckhoff_EQ2xxx.Beckhoff_EQ2xxxEK1122.A_0007_EQ2339_0022_0018.Channel_14.Input <-> Channel 14/Input
//     PlcTask Inputs/GVL_iXlinker.EtherCAT_Master_EQxxxx.Beckhoff_EQ2xxx.Beckhoff_EQ2xxxEK1122.A_0007_EQ2339_0022_0018.Channel_15.Input <-> Channel 15/Input
//     PlcTask Inputs/GVL_iXlinker.EtherCAT_Master_EQxxxx.Beckhoff_EQ2xxx.Beckhoff_EQ2xxxEK1122.A_0007_EQ2339_0022_0018.Channel_16.Input <-> Channel 16/Input
//     PlcTask Outputs/GVL_iXlinker.EtherCAT_Master_EQxxxx.Beckhoff_EQ2xxx.Beckhoff_EQ2xxxEK1122.A_0007_EQ2339_0022_0018.Channel_17.Output <-> Channel 17/Output
//     PlcTask Outputs/GVL_iXlinker.EtherCAT_Master_EQxxxx.Beckhoff_EQ2xxx.Beckhoff_EQ2xxxEK1122.A_0007_EQ2339_0022_0018.Channel_18.Output <-> Channel 18/Output
//     PlcTask Outputs/GVL_iXlinker.EtherCAT_Master_EQxxxx.Beckhoff_EQ2xxx.Beckhoff_EQ2xxxEK1122.A_0007_EQ2339_0022_0018.Channel_19.Output <-> Channel 19/Output
//     PlcTask Outputs/GVL_iXlinker.EtherCAT_Master_EQxxxx.Beckhoff_EQ2xxx.Beckhoff_EQ2xxxEK1122.A_0007_EQ2339_0022_0018.Channel_20.Output <-> Channel 20/Output
//     PlcTask Outputs/GVL_iXlinker.EtherCAT_Master_EQxxxx.Beckhoff_EQ2xxx.Beckhoff_EQ2xxxEK1122.A_0007_EQ2339_0022_0018.Channel_21.Output <-> Channel 21/Output
//     PlcTask Outputs/GVL_iXlinker.EtherCAT_Master_EQxxxx.Beckhoff_EQ2xxx.Beckhoff_EQ2xxxEK1122.A_0007_EQ2339_0022_0018.Channel_22.Output <-> Channel 22/Output
//     PlcTask Outputs/GVL_iXlinker.EtherCAT_Master_EQxxxx.Beckhoff_EQ2xxx.Beckhoff_EQ2xxxEK1122.A_0007_EQ2339_0022_0018.Channel_23.Output <-> Channel 23/Output
//     PlcTask Outputs/GVL_iXlinker.EtherCAT_Master_EQxxxx.Beckhoff_EQ2xxx.Beckhoff_EQ2xxxEK1122.A_0007_EQ2339_0022_0018.Channel_24.Output <-> Channel 24/Output
//     PlcTask Outputs/GVL_iXlinker.EtherCAT_Master_EQxxxx.Beckhoff_EQ2xxx.Beckhoff_EQ2xxxEK1122.A_0007_EQ2339_0022_0018.Channel_25.Output <-> Channel 25/Output
//     PlcTask Outputs/GVL_iXlinker.EtherCAT_Master_EQxxxx.Beckhoff_EQ2xxx.Beckhoff_EQ2xxxEK1122.A_0007_EQ2339_0022_0018.Channel_26.Output <-> Channel 26/Output
//     PlcTask Outputs/GVL_iXlinker.EtherCAT_Master_EQxxxx.Beckhoff_EQ2xxx.Beckhoff_EQ2xxxEK1122.A_0007_EQ2339_0022_0018.Channel_27.Output <-> Channel 27/Output
//     PlcTask Outputs/GVL_iXlinker.EtherCAT_Master_EQxxxx.Beckhoff_EQ2xxx.Beckhoff_EQ2xxxEK1122.A_0007_EQ2339_0022_0018.Channel_28.Output <-> Channel 28/Output
//     PlcTask Outputs/GVL_iXlinker.EtherCAT_Master_EQxxxx.Beckhoff_EQ2xxx.Beckhoff_EQ2xxxEK1122.A_0007_EQ2339_0022_0018.Channel_29.Output <-> Channel 29/Output
//     PlcTask Outputs/GVL_iXlinker.EtherCAT_Master_EQxxxx.Beckhoff_EQ2xxx.Beckhoff_EQ2xxxEK1122.A_0007_EQ2339_0022_0018.Channel_30.Output <-> Channel 30/Output
//     PlcTask Outputs/GVL_iXlinker.EtherCAT_Master_EQxxxx.Beckhoff_EQ2xxx.Beckhoff_EQ2xxxEK1122.A_0007_EQ2339_0022_0018.Channel_31.Output <-> Channel 31/Output
//     PlcTask Outputs/GVL_iXlinker.EtherCAT_Master_EQxxxx.Beckhoff_EQ2xxx.Beckhoff_EQ2xxxEK1122.A_0007_EQ2339_0022_0018.Channel_32.Output <-> Channel 32/Output
//     PlcTask Inputs/GVL_iXlinker.EtherCAT_Master_EQxxxx.Beckhoff_EQ2xxx.Beckhoff_EQ2xxxEK1122.A_0007_EQ2339_0022_0018.WcState.WcState <-> WcState/WcState
//     PlcTask Inputs/GVL_iXlinker.EtherCAT_Master_EQxxxx.Beckhoff_EQ2xxx.Beckhoff_EQ2xxxEK1122.A_0007_EQ2339_0022_0018.WcState.InputToggle <-> WcState/InputToggle
//     PlcTask Inputs/GVL_iXlinker.EtherCAT_Master_EQxxxx.Beckhoff_EQ2xxx.Beckhoff_EQ2xxxEK1122.A_0007_EQ2339_0022_0018.InfoData.State <-> InfoData/State
//   PLC/PLC Instance <-> EtherCAT Master EQxxxx/Beckhoff EQ2xxx/Beckhoff EQ2xxxEK1122/A_0008(EQ2339-0022-0019)
//     PlcTask Inputs/GVL_iXlinker.EtherCAT_Master_EQxxxx.Beckhoff_EQ2xxx.Beckhoff_EQ2xxxEK1122.A_0008_EQ2339_0022_0019.Channel_1.Input <-> Channel 1/Input
//     PlcTask Inputs/GVL_iXlinker.EtherCAT_Master_EQxxxx.Beckhoff_EQ2xxx.Beckhoff_EQ2xxxEK1122.A_0008_EQ2339_0022_0019.Channel_2.Input <-> Channel 2/Input
//     PlcTask Inputs/GVL_iXlinker.EtherCAT_Master_EQxxxx.Beckhoff_EQ2xxx.Beckhoff_EQ2xxxEK1122.A_0008_EQ2339_0022_0019.Channel_3.Input <-> Channel 3/Input
//     PlcTask Inputs/GVL_iXlinker.EtherCAT_Master_EQxxxx.Beckhoff_EQ2xxx.Beckhoff_EQ2xxxEK1122.A_0008_EQ2339_0022_0019.Channel_4.Input <-> Channel 4/Input
//     PlcTask Inputs/GVL_iXlinker.EtherCAT_Master_EQxxxx.Beckhoff_EQ2xxx.Beckhoff_EQ2xxxEK1122.A_0008_EQ2339_0022_0019.Channel_5.Input <-> Channel 5/Input
//     PlcTask Inputs/GVL_iXlinker.EtherCAT_Master_EQxxxx.Beckhoff_EQ2xxx.Beckhoff_EQ2xxxEK1122.A_0008_EQ2339_0022_0019.Channel_6.Input <-> Channel 6/Input
//     PlcTask Inputs/GVL_iXlinker.EtherCAT_Master_EQxxxx.Beckhoff_EQ2xxx.Beckhoff_EQ2xxxEK1122.A_0008_EQ2339_0022_0019.Channel_7.Input <-> Channel 7/Input
//     PlcTask Inputs/GVL_iXlinker.EtherCAT_Master_EQxxxx.Beckhoff_EQ2xxx.Beckhoff_EQ2xxxEK1122.A_0008_EQ2339_0022_0019.Channel_8.Input <-> Channel 8/Input
//     PlcTask Inputs/GVL_iXlinker.EtherCAT_Master_EQxxxx.Beckhoff_EQ2xxx.Beckhoff_EQ2xxxEK1122.A_0008_EQ2339_0022_0019.Channel_9.Input <-> Channel 9/Input
//     PlcTask Inputs/GVL_iXlinker.EtherCAT_Master_EQxxxx.Beckhoff_EQ2xxx.Beckhoff_EQ2xxxEK1122.A_0008_EQ2339_0022_0019.Channel_10.Input <-> Channel 10/Input
//     PlcTask Inputs/GVL_iXlinker.EtherCAT_Master_EQxxxx.Beckhoff_EQ2xxx.Beckhoff_EQ2xxxEK1122.A_0008_EQ2339_0022_0019.Channel_11.Input <-> Channel 11/Input
//     PlcTask Inputs/GVL_iXlinker.EtherCAT_Master_EQxxxx.Beckhoff_EQ2xxx.Beckhoff_EQ2xxxEK1122.A_0008_EQ2339_0022_0019.Channel_12.Input <-> Channel 12/Input
//     PlcTask Inputs/GVL_iXlinker.EtherCAT_Master_EQxxxx.Beckhoff_EQ2xxx.Beckhoff_EQ2xxxEK1122.A_0008_EQ2339_0022_0019.Channel_13.Input <-> Channel 13/Input
//     PlcTask Inputs/GVL_iXlinker.EtherCAT_Master_EQxxxx.Beckhoff_EQ2xxx.Beckhoff_EQ2xxxEK1122.A_0008_EQ2339_0022_0019.Channel_14.Input <-> Channel 14/Input
//     PlcTask Inputs/GVL_iXlinker.EtherCAT_Master_EQxxxx.Beckhoff_EQ2xxx.Beckhoff_EQ2xxxEK1122.A_0008_EQ2339_0022_0019.Channel_15.Input <-> Channel 15/Input
//     PlcTask Inputs/GVL_iXlinker.EtherCAT_Master_EQxxxx.Beckhoff_EQ2xxx.Beckhoff_EQ2xxxEK1122.A_0008_EQ2339_0022_0019.Channel_16.Input <-> Channel 16/Input
//     PlcTask Outputs/GVL_iXlinker.EtherCAT_Master_EQxxxx.Beckhoff_EQ2xxx.Beckhoff_EQ2xxxEK1122.A_0008_EQ2339_0022_0019.Channel_17.Output <-> Channel 17/Output
//     PlcTask Outputs/GVL_iXlinker.EtherCAT_Master_EQxxxx.Beckhoff_EQ2xxx.Beckhoff_EQ2xxxEK1122.A_0008_EQ2339_0022_0019.Channel_18.Output <-> Channel 18/Output
//     PlcTask Outputs/GVL_iXlinker.EtherCAT_Master_EQxxxx.Beckhoff_EQ2xxx.Beckhoff_EQ2xxxEK1122.A_0008_EQ2339_0022_0019.Channel_19.Output <-> Channel 19/Output
//     PlcTask Outputs/GVL_iXlinker.EtherCAT_Master_EQxxxx.Beckhoff_EQ2xxx.Beckhoff_EQ2xxxEK1122.A_0008_EQ2339_0022_0019.Channel_20.Output <-> Channel 20/Output
//     PlcTask Outputs/GVL_iXlinker.EtherCAT_Master_EQxxxx.Beckhoff_EQ2xxx.Beckhoff_EQ2xxxEK1122.A_0008_EQ2339_0022_0019.Channel_21.Output <-> Channel 21/Output
//     PlcTask Outputs/GVL_iXlinker.EtherCAT_Master_EQxxxx.Beckhoff_EQ2xxx.Beckhoff_EQ2xxxEK1122.A_0008_EQ2339_0022_0019.Channel_22.Output <-> Channel 22/Output
//     PlcTask Outputs/GVL_iXlinker.EtherCAT_Master_EQxxxx.Beckhoff_EQ2xxx.Beckhoff_EQ2xxxEK1122.A_0008_EQ2339_0022_0019.Channel_23.Output <-> Channel 23/Output
//     PlcTask Outputs/GVL_iXlinker.EtherCAT_Master_EQxxxx.Beckhoff_EQ2xxx.Beckhoff_EQ2xxxEK1122.A_0008_EQ2339_0022_0019.Channel_24.Output <-> Channel 24/Output
//     PlcTask Outputs/GVL_iXlinker.EtherCAT_Master_EQxxxx.Beckhoff_EQ2xxx.Beckhoff_EQ2xxxEK1122.A_0008_EQ2339_0022_0019.Channel_25.Output <-> Channel 25/Output
//     PlcTask Outputs/GVL_iXlinker.EtherCAT_Master_EQxxxx.Beckhoff_EQ2xxx.Beckhoff_EQ2xxxEK1122.A_0008_EQ2339_0022_0019.Channel_26.Output <-> Channel 26/Output
//     PlcTask Outputs/GVL_iXlinker.EtherCAT_Master_EQxxxx.Beckhoff_EQ2xxx.Beckhoff_EQ2xxxEK1122.A_0008_EQ2339_0022_0019.Channel_27.Output <-> Channel 27/Output
//     PlcTask Outputs/GVL_iXlinker.EtherCAT_Master_EQxxxx.Beckhoff_EQ2xxx.Beckhoff_EQ2xxxEK1122.A_0008_EQ2339_0022_0019.Channel_28.Output <-> Channel 28/Output
//     PlcTask Outputs/GVL_iXlinker.EtherCAT_Master_EQxxxx.Beckhoff_EQ2xxx.Beckhoff_EQ2xxxEK1122.A_0008_EQ2339_0022_0019.Channel_29.Output <-> Channel 29/Output
//     PlcTask Outputs/GVL_iXlinker.EtherCAT_Master_EQxxxx.Beckhoff_EQ2xxx.Beckhoff_EQ2xxxEK1122.A_0008_EQ2339_0022_0019.Channel_30.Output <-> Channel 30/Output
//     PlcTask Outputs/GVL_iXlinker.EtherCAT_Master_EQxxxx.Beckhoff_EQ2xxx.Beckhoff_EQ2xxxEK1122.A_0008_EQ2339_0022_0019.Channel_31.Output <-> Channel 31/Output
//     PlcTask Outputs/GVL_iXlinker.EtherCAT_Master_EQxxxx.Beckhoff_EQ2xxx.Beckhoff_EQ2xxxEK1122.A_0008_EQ2339_0022_0019.Channel_32.Output <-> Channel 32/Output
//     PlcTask Inputs/GVL_iXlinker.EtherCAT_Master_EQxxxx.Beckhoff_EQ2xxx.Beckhoff_EQ2xxxEK1122.A_0008_EQ2339_0022_0019.WcState.WcState <-> WcState/WcState
//     PlcTask Inputs/GVL_iXlinker.EtherCAT_Master_EQxxxx.Beckhoff_EQ2xxx.Beckhoff_EQ2xxxEK1122.A_0008_EQ2339_0022_0019.WcState.InputToggle <-> WcState/InputToggle
//     PlcTask Inputs/GVL_iXlinker.EtherCAT_Master_EQxxxx.Beckhoff_EQ2xxx.Beckhoff_EQ2xxxEK1122.A_0008_EQ2339_0022_0019.InfoData.State <-> InfoData/State
//   PLC/PLC Instance <-> EtherCAT Master EQxxxx/Beckhoff EQ2xxx/Beckhoff EQ2xxxEK1122/A_0009(EQ2809-0022-0016)
//     PlcTask Outputs/GVL_iXlinker.EtherCAT_Master_EQxxxx.Beckhoff_EQ2xxx.Beckhoff_EQ2xxxEK1122.A_0009_EQ2809_0022_0016.Channel_1.Output <-> Channel 1/Output
//     PlcTask Outputs/GVL_iXlinker.EtherCAT_Master_EQxxxx.Beckhoff_EQ2xxx.Beckhoff_EQ2xxxEK1122.A_0009_EQ2809_0022_0016.Channel_2.Output <-> Channel 2/Output
//     PlcTask Outputs/GVL_iXlinker.EtherCAT_Master_EQxxxx.Beckhoff_EQ2xxx.Beckhoff_EQ2xxxEK1122.A_0009_EQ2809_0022_0016.Channel_3.Output <-> Channel 3/Output
//     PlcTask Outputs/GVL_iXlinker.EtherCAT_Master_EQxxxx.Beckhoff_EQ2xxx.Beckhoff_EQ2xxxEK1122.A_0009_EQ2809_0022_0016.Channel_4.Output <-> Channel 4/Output
//     PlcTask Outputs/GVL_iXlinker.EtherCAT_Master_EQxxxx.Beckhoff_EQ2xxx.Beckhoff_EQ2xxxEK1122.A_0009_EQ2809_0022_0016.Channel_5.Output <-> Channel 5/Output
//     PlcTask Outputs/GVL_iXlinker.EtherCAT_Master_EQxxxx.Beckhoff_EQ2xxx.Beckhoff_EQ2xxxEK1122.A_0009_EQ2809_0022_0016.Channel_6.Output <-> Channel 6/Output
//     PlcTask Outputs/GVL_iXlinker.EtherCAT_Master_EQxxxx.Beckhoff_EQ2xxx.Beckhoff_EQ2xxxEK1122.A_0009_EQ2809_0022_0016.Channel_7.Output <-> Channel 7/Output
//     PlcTask Outputs/GVL_iXlinker.EtherCAT_Master_EQxxxx.Beckhoff_EQ2xxx.Beckhoff_EQ2xxxEK1122.A_0009_EQ2809_0022_0016.Channel_8.Output <-> Channel 8/Output
//     PlcTask Outputs/GVL_iXlinker.EtherCAT_Master_EQxxxx.Beckhoff_EQ2xxx.Beckhoff_EQ2xxxEK1122.A_0009_EQ2809_0022_0016.Channel_9.Output <-> Channel 9/Output
//     PlcTask Outputs/GVL_iXlinker.EtherCAT_Master_EQxxxx.Beckhoff_EQ2xxx.Beckhoff_EQ2xxxEK1122.A_0009_EQ2809_0022_0016.Channel_10.Output <-> Channel 10/Output
//     PlcTask Outputs/GVL_iXlinker.EtherCAT_Master_EQxxxx.Beckhoff_EQ2xxx.Beckhoff_EQ2xxxEK1122.A_0009_EQ2809_0022_0016.Channel_11.Output <-> Channel 11/Output
//     PlcTask Outputs/GVL_iXlinker.EtherCAT_Master_EQxxxx.Beckhoff_EQ2xxx.Beckhoff_EQ2xxxEK1122.A_0009_EQ2809_0022_0016.Channel_12.Output <-> Channel 12/Output
//     PlcTask Outputs/GVL_iXlinker.EtherCAT_Master_EQxxxx.Beckhoff_EQ2xxx.Beckhoff_EQ2xxxEK1122.A_0009_EQ2809_0022_0016.Channel_13.Output <-> Channel 13/Output
//     PlcTask Outputs/GVL_iXlinker.EtherCAT_Master_EQxxxx.Beckhoff_EQ2xxx.Beckhoff_EQ2xxxEK1122.A_0009_EQ2809_0022_0016.Channel_14.Output <-> Channel 14/Output
//     PlcTask Outputs/GVL_iXlinker.EtherCAT_Master_EQxxxx.Beckhoff_EQ2xxx.Beckhoff_EQ2xxxEK1122.A_0009_EQ2809_0022_0016.Channel_15.Output <-> Channel 15/Output
//     PlcTask Outputs/GVL_iXlinker.EtherCAT_Master_EQxxxx.Beckhoff_EQ2xxx.Beckhoff_EQ2xxxEK1122.A_0009_EQ2809_0022_0016.Channel_16.Output <-> Channel 16/Output
//     PlcTask Inputs/GVL_iXlinker.EtherCAT_Master_EQxxxx.Beckhoff_EQ2xxx.Beckhoff_EQ2xxxEK1122.A_0009_EQ2809_0022_0016.WcState.WcState <-> WcState/WcState
//     PlcTask Inputs/GVL_iXlinker.EtherCAT_Master_EQxxxx.Beckhoff_EQ2xxx.Beckhoff_EQ2xxxEK1122.A_0009_EQ2809_0022_0016.InfoData.State <-> InfoData/State
//   PLC/PLC Instance <-> EtherCAT Master EQxxxx/Beckhoff EQ2xxx/Beckhoff EQ2xxxEK1122/A_0010(EQ2809-0022-0017)
//     PlcTask Outputs/GVL_iXlinker.EtherCAT_Master_EQxxxx.Beckhoff_EQ2xxx.Beckhoff_EQ2xxxEK1122.A_0010_EQ2809_0022_0017.Channel_1.Output <-> Channel 1/Output
//     PlcTask Outputs/GVL_iXlinker.EtherCAT_Master_EQxxxx.Beckhoff_EQ2xxx.Beckhoff_EQ2xxxEK1122.A_0010_EQ2809_0022_0017.Channel_2.Output <-> Channel 2/Output
//     PlcTask Outputs/GVL_iXlinker.EtherCAT_Master_EQxxxx.Beckhoff_EQ2xxx.Beckhoff_EQ2xxxEK1122.A_0010_EQ2809_0022_0017.Channel_3.Output <-> Channel 3/Output
//     PlcTask Outputs/GVL_iXlinker.EtherCAT_Master_EQxxxx.Beckhoff_EQ2xxx.Beckhoff_EQ2xxxEK1122.A_0010_EQ2809_0022_0017.Channel_4.Output <-> Channel 4/Output
//     PlcTask Outputs/GVL_iXlinker.EtherCAT_Master_EQxxxx.Beckhoff_EQ2xxx.Beckhoff_EQ2xxxEK1122.A_0010_EQ2809_0022_0017.Channel_5.Output <-> Channel 5/Output
//     PlcTask Outputs/GVL_iXlinker.EtherCAT_Master_EQxxxx.Beckhoff_EQ2xxx.Beckhoff_EQ2xxxEK1122.A_0010_EQ2809_0022_0017.Channel_6.Output <-> Channel 6/Output
//     PlcTask Outputs/GVL_iXlinker.EtherCAT_Master_EQxxxx.Beckhoff_EQ2xxx.Beckhoff_EQ2xxxEK1122.A_0010_EQ2809_0022_0017.Channel_7.Output <-> Channel 7/Output
//     PlcTask Outputs/GVL_iXlinker.EtherCAT_Master_EQxxxx.Beckhoff_EQ2xxx.Beckhoff_EQ2xxxEK1122.A_0010_EQ2809_0022_0017.Channel_8.Output <-> Channel 8/Output
//     PlcTask Outputs/GVL_iXlinker.EtherCAT_Master_EQxxxx.Beckhoff_EQ2xxx.Beckhoff_EQ2xxxEK1122.A_0010_EQ2809_0022_0017.Channel_9.Output <-> Channel 9/Output
//     PlcTask Outputs/GVL_iXlinker.EtherCAT_Master_EQxxxx.Beckhoff_EQ2xxx.Beckhoff_EQ2xxxEK1122.A_0010_EQ2809_0022_0017.Channel_10.Output <-> Channel 10/Output
//     PlcTask Outputs/GVL_iXlinker.EtherCAT_Master_EQxxxx.Beckhoff_EQ2xxx.Beckhoff_EQ2xxxEK1122.A_0010_EQ2809_0022_0017.Channel_11.Output <-> Channel 11/Output
//     PlcTask Outputs/GVL_iXlinker.EtherCAT_Master_EQxxxx.Beckhoff_EQ2xxx.Beckhoff_EQ2xxxEK1122.A_0010_EQ2809_0022_0017.Channel_12.Output <-> Channel 12/Output
//     PlcTask Outputs/GVL_iXlinker.EtherCAT_Master_EQxxxx.Beckhoff_EQ2xxx.Beckhoff_EQ2xxxEK1122.A_0010_EQ2809_0022_0017.Channel_13.Output <-> Channel 13/Output
//     PlcTask Outputs/GVL_iXlinker.EtherCAT_Master_EQxxxx.Beckhoff_EQ2xxx.Beckhoff_EQ2xxxEK1122.A_0010_EQ2809_0022_0017.Channel_14.Output <-> Channel 14/Output
//     PlcTask Outputs/GVL_iXlinker.EtherCAT_Master_EQxxxx.Beckhoff_EQ2xxx.Beckhoff_EQ2xxxEK1122.A_0010_EQ2809_0022_0017.Channel_15.Output <-> Channel 15/Output
//     PlcTask Outputs/GVL_iXlinker.EtherCAT_Master_EQxxxx.Beckhoff_EQ2xxx.Beckhoff_EQ2xxxEK1122.A_0010_EQ2809_0022_0017.Channel_16.Output <-> Channel 16/Output
//     PlcTask Inputs/GVL_iXlinker.EtherCAT_Master_EQxxxx.Beckhoff_EQ2xxx.Beckhoff_EQ2xxxEK1122.A_0010_EQ2809_0022_0017.WcState.WcState <-> WcState/WcState
//     PlcTask Inputs/GVL_iXlinker.EtherCAT_Master_EQxxxx.Beckhoff_EQ2xxx.Beckhoff_EQ2xxxEK1122.A_0010_EQ2809_0022_0017.InfoData.State <-> InfoData/State
//   PLC/PLC Instance <-> EtherCAT Master EQxxxx/Beckhoff EQ2xxx/Beckhoff EQ2xxxEK1122/A_0011(EQ2809-0022-0018)
//     PlcTask Outputs/GVL_iXlinker.EtherCAT_Master_EQxxxx.Beckhoff_EQ2xxx.Beckhoff_EQ2xxxEK1122.A_0011_EQ2809_0022_0018.Channel_1.Output <-> Channel 1/Output
//     PlcTask Outputs/GVL_iXlinker.EtherCAT_Master_EQxxxx.Beckhoff_EQ2xxx.Beckhoff_EQ2xxxEK1122.A_0011_EQ2809_0022_0018.Channel_2.Output <-> Channel 2/Output
//     PlcTask Outputs/GVL_iXlinker.EtherCAT_Master_EQxxxx.Beckhoff_EQ2xxx.Beckhoff_EQ2xxxEK1122.A_0011_EQ2809_0022_0018.Channel_3.Output <-> Channel 3/Output
//     PlcTask Outputs/GVL_iXlinker.EtherCAT_Master_EQxxxx.Beckhoff_EQ2xxx.Beckhoff_EQ2xxxEK1122.A_0011_EQ2809_0022_0018.Channel_4.Output <-> Channel 4/Output
//     PlcTask Outputs/GVL_iXlinker.EtherCAT_Master_EQxxxx.Beckhoff_EQ2xxx.Beckhoff_EQ2xxxEK1122.A_0011_EQ2809_0022_0018.Channel_5.Output <-> Channel 5/Output
//     PlcTask Outputs/GVL_iXlinker.EtherCAT_Master_EQxxxx.Beckhoff_EQ2xxx.Beckhoff_EQ2xxxEK1122.A_0011_EQ2809_0022_0018.Channel_6.Output <-> Channel 6/Output
//     PlcTask Outputs/GVL_iXlinker.EtherCAT_Master_EQxxxx.Beckhoff_EQ2xxx.Beckhoff_EQ2xxxEK1122.A_0011_EQ2809_0022_0018.Channel_7.Output <-> Channel 7/Output
//     PlcTask Outputs/GVL_iXlinker.EtherCAT_Master_EQxxxx.Beckhoff_EQ2xxx.Beckhoff_EQ2xxxEK1122.A_0011_EQ2809_0022_0018.Channel_8.Output <-> Channel 8/Output
//     PlcTask Outputs/GVL_iXlinker.EtherCAT_Master_EQxxxx.Beckhoff_EQ2xxx.Beckhoff_EQ2xxxEK1122.A_0011_EQ2809_0022_0018.Channel_9.Output <-> Channel 9/Output
//     PlcTask Outputs/GVL_iXlinker.EtherCAT_Master_EQxxxx.Beckhoff_EQ2xxx.Beckhoff_EQ2xxxEK1122.A_0011_EQ2809_0022_0018.Channel_10.Output <-> Channel 10/Output
//     PlcTask Outputs/GVL_iXlinker.EtherCAT_Master_EQxxxx.Beckhoff_EQ2xxx.Beckhoff_EQ2xxxEK1122.A_0011_EQ2809_0022_0018.Channel_11.Output <-> Channel 11/Output
//     PlcTask Outputs/GVL_iXlinker.EtherCAT_Master_EQxxxx.Beckhoff_EQ2xxx.Beckhoff_EQ2xxxEK1122.A_0011_EQ2809_0022_0018.Channel_12.Output <-> Channel 12/Output
//     PlcTask Outputs/GVL_iXlinker.EtherCAT_Master_EQxxxx.Beckhoff_EQ2xxx.Beckhoff_EQ2xxxEK1122.A_0011_EQ2809_0022_0018.Channel_13.Output <-> Channel 13/Output
//     PlcTask Outputs/GVL_iXlinker.EtherCAT_Master_EQxxxx.Beckhoff_EQ2xxx.Beckhoff_EQ2xxxEK1122.A_0011_EQ2809_0022_0018.Channel_14.Output <-> Channel 14/Output
//     PlcTask Outputs/GVL_iXlinker.EtherCAT_Master_EQxxxx.Beckhoff_EQ2xxx.Beckhoff_EQ2xxxEK1122.A_0011_EQ2809_0022_0018.Channel_15.Output <-> Channel 15/Output
//     PlcTask Outputs/GVL_iXlinker.EtherCAT_Master_EQxxxx.Beckhoff_EQ2xxx.Beckhoff_EQ2xxxEK1122.A_0011_EQ2809_0022_0018.Channel_16.Output <-> Channel 16/Output
//     PlcTask Inputs/GVL_iXlinker.EtherCAT_Master_EQxxxx.Beckhoff_EQ2xxx.Beckhoff_EQ2xxxEK1122.A_0011_EQ2809_0022_0018.WcState.WcState <-> WcState/WcState
//     PlcTask Inputs/GVL_iXlinker.EtherCAT_Master_EQxxxx.Beckhoff_EQ2xxx.Beckhoff_EQ2xxxEK1122.A_0011_EQ2809_0022_0018.InfoData.State <-> InfoData/State
//   PLC/PLC Instance <-> EtherCAT Master EQxxxx/Beckhoff EQ3xxx
//     PlcTask Inputs/GVL_iXlinker.EtherCAT_Master_EQxxxx.Beckhoff_EQ3xxx.InfoData.State <-> InfoData/State
//   PLC/PLC Instance <-> EtherCAT Master EQxxxx/Beckhoff EQ3xxx/Beckhoff EQ3xxxEK1122
//     PlcTask Inputs/GVL_iXlinker.EtherCAT_Master_EQxxxx.Beckhoff_EQ3xxx.Beckhoff_EQ3xxxEK1122.InfoData.State <-> InfoData/State
//   PLC/PLC Instance <-> EtherCAT Master EQxxxx/Beckhoff EQ3xxx/Beckhoff EQ3xxxEK1122/Beckhoff EQ3xxxsub EK1100
//     PlcTask Inputs/GVL_iXlinker.EtherCAT_Master_EQxxxx.Beckhoff_EQ3xxx.Beckhoff_EQ3xxxEK1122.Beckhoff_EQ3xxxsub_EK1100.InfoData.State <-> InfoData/State
//   PLC/PLC Instance <-> EtherCAT Master EQxxxx/Beckhoff EQ3xxx/Beckhoff EQ3xxxEK1122/A_0001(EQ3174-0002-0016)
//     PlcTask Inputs/GVL_iXlinker.EtherCAT_Master_EQxxxx.Beckhoff_EQ3xxx.Beckhoff_EQ3xxxEK1122.A_0001_EQ3174_0002_0016.AI_Standard_Channel_1.Status/Underrange <-> AI Standard Channel 1/Status/Underrange
//     PlcTask Inputs/GVL_iXlinker.EtherCAT_Master_EQxxxx.Beckhoff_EQ3xxx.Beckhoff_EQ3xxxEK1122.A_0001_EQ3174_0002_0016.AI_Standard_Channel_2.Status/Underrange <-> AI Standard Channel 2/Status/Underrange
//     PlcTask Inputs/GVL_iXlinker.EtherCAT_Master_EQxxxx.Beckhoff_EQ3xxx.Beckhoff_EQ3xxxEK1122.A_0001_EQ3174_0002_0016.AI_Standard_Channel_3.Status/Underrange <-> AI Standard Channel 3/Status/Underrange
//     PlcTask Inputs/GVL_iXlinker.EtherCAT_Master_EQxxxx.Beckhoff_EQ3xxx.Beckhoff_EQ3xxxEK1122.A_0001_EQ3174_0002_0016.AI_Standard_Channel_4.Status/Underrange <-> AI Standard Channel 4/Status/Underrange
//     PlcTask Inputs/GVL_iXlinker.EtherCAT_Master_EQxxxx.Beckhoff_EQ3xxx.Beckhoff_EQ3xxxEK1122.A_0001_EQ3174_0002_0016.AI_Standard_Channel_1.Status/Overrange <-> AI Standard Channel 1/Status/Overrange
//     PlcTask Inputs/GVL_iXlinker.EtherCAT_Master_EQxxxx.Beckhoff_EQ3xxx.Beckhoff_EQ3xxxEK1122.A_0001_EQ3174_0002_0016.AI_Standard_Channel_2.Status/Overrange <-> AI Standard Channel 2/Status/Overrange
//     PlcTask Inputs/GVL_iXlinker.EtherCAT_Master_EQxxxx.Beckhoff_EQ3xxx.Beckhoff_EQ3xxxEK1122.A_0001_EQ3174_0002_0016.AI_Standard_Channel_3.Status/Overrange <-> AI Standard Channel 3/Status/Overrange
//     PlcTask Inputs/GVL_iXlinker.EtherCAT_Master_EQxxxx.Beckhoff_EQ3xxx.Beckhoff_EQ3xxxEK1122.A_0001_EQ3174_0002_0016.AI_Standard_Channel_4.Status/Overrange <-> AI Standard Channel 4/Status/Overrange
//     PlcTask Inputs/GVL_iXlinker.EtherCAT_Master_EQxxxx.Beckhoff_EQ3xxx.Beckhoff_EQ3xxxEK1122.A_0001_EQ3174_0002_0016.AI_Standard_Channel_1.Status/Limit_1 <-> AI Standard Channel 1/Status/Limit 1
//     PlcTask Inputs/GVL_iXlinker.EtherCAT_Master_EQxxxx.Beckhoff_EQ3xxx.Beckhoff_EQ3xxxEK1122.A_0001_EQ3174_0002_0016.AI_Standard_Channel_1.Status/Limit_2 <-> AI Standard Channel 1/Status/Limit 2
//     PlcTask Inputs/GVL_iXlinker.EtherCAT_Master_EQxxxx.Beckhoff_EQ3xxx.Beckhoff_EQ3xxxEK1122.A_0001_EQ3174_0002_0016.AI_Standard_Channel_2.Status/Limit_1 <-> AI Standard Channel 2/Status/Limit 1
//     PlcTask Inputs/GVL_iXlinker.EtherCAT_Master_EQxxxx.Beckhoff_EQ3xxx.Beckhoff_EQ3xxxEK1122.A_0001_EQ3174_0002_0016.AI_Standard_Channel_2.Status/Limit_2 <-> AI Standard Channel 2/Status/Limit 2
//     PlcTask Inputs/GVL_iXlinker.EtherCAT_Master_EQxxxx.Beckhoff_EQ3xxx.Beckhoff_EQ3xxxEK1122.A_0001_EQ3174_0002_0016.AI_Standard_Channel_3.Status/Limit_1 <-> AI Standard Channel 3/Status/Limit 1
//     PlcTask Inputs/GVL_iXlinker.EtherCAT_Master_EQxxxx.Beckhoff_EQ3xxx.Beckhoff_EQ3xxxEK1122.A_0001_EQ3174_0002_0016.AI_Standard_Channel_3.Status/Limit_2 <-> AI Standard Channel 3/Status/Limit 2
//     PlcTask Inputs/GVL_iXlinker.EtherCAT_Master_EQxxxx.Beckhoff_EQ3xxx.Beckhoff_EQ3xxxEK1122.A_0001_EQ3174_0002_0016.AI_Standard_Channel_4.Status/Limit_1 <-> AI Standard Channel 4/Status/Limit 1
//     PlcTask Inputs/GVL_iXlinker.EtherCAT_Master_EQxxxx.Beckhoff_EQ3xxx.Beckhoff_EQ3xxxEK1122.A_0001_EQ3174_0002_0016.AI_Standard_Channel_4.Status/Limit_2 <-> AI Standard Channel 4/Status/Limit 2
//     PlcTask Inputs/GVL_iXlinker.EtherCAT_Master_EQxxxx.Beckhoff_EQ3xxx.Beckhoff_EQ3xxxEK1122.A_0001_EQ3174_0002_0016.AI_Standard_Channel_1.Status/Error <-> AI Standard Channel 1/Status/Error
//     PlcTask Inputs/GVL_iXlinker.EtherCAT_Master_EQxxxx.Beckhoff_EQ3xxx.Beckhoff_EQ3xxxEK1122.A_0001_EQ3174_0002_0016.AI_Standard_Channel_2.Status/Error <-> AI Standard Channel 2/Status/Error
//     PlcTask Inputs/GVL_iXlinker.EtherCAT_Master_EQxxxx.Beckhoff_EQ3xxx.Beckhoff_EQ3xxxEK1122.A_0001_EQ3174_0002_0016.AI_Standard_Channel_3.Status/Error <-> AI Standard Channel 3/Status/Error
//     PlcTask Inputs/GVL_iXlinker.EtherCAT_Master_EQxxxx.Beckhoff_EQ3xxx.Beckhoff_EQ3xxxEK1122.A_0001_EQ3174_0002_0016.AI_Standard_Channel_4.Status/Error <-> AI Standard Channel 4/Status/Error
//     PlcTask Inputs/GVL_iXlinker.EtherCAT_Master_EQxxxx.Beckhoff_EQ3xxx.Beckhoff_EQ3xxxEK1122.A_0001_EQ3174_0002_0016.AI_Standard_Channel_1.Status/Sync_error <-> AI Standard Channel 1/Status/Sync error
//     PlcTask Inputs/GVL_iXlinker.EtherCAT_Master_EQxxxx.Beckhoff_EQ3xxx.Beckhoff_EQ3xxxEK1122.A_0001_EQ3174_0002_0016.AI_Standard_Channel_2.Status/Sync_error <-> AI Standard Channel 2/Status/Sync error
//     PlcTask Inputs/GVL_iXlinker.EtherCAT_Master_EQxxxx.Beckhoff_EQ3xxx.Beckhoff_EQ3xxxEK1122.A_0001_EQ3174_0002_0016.AI_Standard_Channel_3.Status/Sync_error <-> AI Standard Channel 3/Status/Sync error
//     PlcTask Inputs/GVL_iXlinker.EtherCAT_Master_EQxxxx.Beckhoff_EQ3xxx.Beckhoff_EQ3xxxEK1122.A_0001_EQ3174_0002_0016.AI_Standard_Channel_4.Status/Sync_error <-> AI Standard Channel 4/Status/Sync error
//     PlcTask Inputs/GVL_iXlinker.EtherCAT_Master_EQxxxx.Beckhoff_EQ3xxx.Beckhoff_EQ3xxxEK1122.A_0001_EQ3174_0002_0016.AI_Standard_Channel_1.Status/TxPDO_State <-> AI Standard Channel 1/Status/TxPDO State
//     PlcTask Inputs/GVL_iXlinker.EtherCAT_Master_EQxxxx.Beckhoff_EQ3xxx.Beckhoff_EQ3xxxEK1122.A_0001_EQ3174_0002_0016.AI_Standard_Channel_2.Status/TxPDO_State <-> AI Standard Channel 2/Status/TxPDO State
//     PlcTask Inputs/GVL_iXlinker.EtherCAT_Master_EQxxxx.Beckhoff_EQ3xxx.Beckhoff_EQ3xxxEK1122.A_0001_EQ3174_0002_0016.AI_Standard_Channel_3.Status/TxPDO_State <-> AI Standard Channel 3/Status/TxPDO State
//     PlcTask Inputs/GVL_iXlinker.EtherCAT_Master_EQxxxx.Beckhoff_EQ3xxx.Beckhoff_EQ3xxxEK1122.A_0001_EQ3174_0002_0016.AI_Standard_Channel_4.Status/TxPDO_State <-> AI Standard Channel 4/Status/TxPDO State
//     PlcTask Inputs/GVL_iXlinker.EtherCAT_Master_EQxxxx.Beckhoff_EQ3xxx.Beckhoff_EQ3xxxEK1122.A_0001_EQ3174_0002_0016.AI_Standard_Channel_1.Status/TxPDO_Toggle <-> AI Standard Channel 1/Status/TxPDO Toggle
//     PlcTask Inputs/GVL_iXlinker.EtherCAT_Master_EQxxxx.Beckhoff_EQ3xxx.Beckhoff_EQ3xxxEK1122.A_0001_EQ3174_0002_0016.AI_Standard_Channel_2.Status/TxPDO_Toggle <-> AI Standard Channel 2/Status/TxPDO Toggle
//     PlcTask Inputs/GVL_iXlinker.EtherCAT_Master_EQxxxx.Beckhoff_EQ3xxx.Beckhoff_EQ3xxxEK1122.A_0001_EQ3174_0002_0016.AI_Standard_Channel_3.Status/TxPDO_Toggle <-> AI Standard Channel 3/Status/TxPDO Toggle
//     PlcTask Inputs/GVL_iXlinker.EtherCAT_Master_EQxxxx.Beckhoff_EQ3xxx.Beckhoff_EQ3xxxEK1122.A_0001_EQ3174_0002_0016.AI_Standard_Channel_4.Status/TxPDO_Toggle <-> AI Standard Channel 4/Status/TxPDO Toggle
//     PlcTask Inputs/GVL_iXlinker.EtherCAT_Master_EQxxxx.Beckhoff_EQ3xxx.Beckhoff_EQ3xxxEK1122.A_0001_EQ3174_0002_0016.AI_Standard_Channel_1.Value <-> AI Standard Channel 1/Value
//     PlcTask Inputs/GVL_iXlinker.EtherCAT_Master_EQxxxx.Beckhoff_EQ3xxx.Beckhoff_EQ3xxxEK1122.A_0001_EQ3174_0002_0016.AI_Standard_Channel_2.Value <-> AI Standard Channel 2/Value
//     PlcTask Inputs/GVL_iXlinker.EtherCAT_Master_EQxxxx.Beckhoff_EQ3xxx.Beckhoff_EQ3xxxEK1122.A_0001_EQ3174_0002_0016.AI_Standard_Channel_3.Value <-> AI Standard Channel 3/Value
//     PlcTask Inputs/GVL_iXlinker.EtherCAT_Master_EQxxxx.Beckhoff_EQ3xxx.Beckhoff_EQ3xxxEK1122.A_0001_EQ3174_0002_0016.AI_Standard_Channel_4.Value <-> AI Standard Channel 4/Value
//     PlcTask Inputs/GVL_iXlinker.EtherCAT_Master_EQxxxx.Beckhoff_EQ3xxx.Beckhoff_EQ3xxxEK1122.A_0001_EQ3174_0002_0016.WcState.WcState <-> WcState/WcState
//     PlcTask Inputs/GVL_iXlinker.EtherCAT_Master_EQxxxx.Beckhoff_EQ3xxx.Beckhoff_EQ3xxxEK1122.A_0001_EQ3174_0002_0016.WcState.InputToggle <-> WcState/InputToggle
//     PlcTask Inputs/GVL_iXlinker.EtherCAT_Master_EQxxxx.Beckhoff_EQ3xxx.Beckhoff_EQ3xxxEK1122.A_0001_EQ3174_0002_0016.InfoData.AdsAddr <-> InfoData/AdsAddr
//     PlcTask Inputs/GVL_iXlinker.EtherCAT_Master_EQxxxx.Beckhoff_EQ3xxx.Beckhoff_EQ3xxxEK1122.A_0001_EQ3174_0002_0016.InfoData.State <-> InfoData/State
//   PLC/PLC Instance <-> EtherCAT Master EQxxxx/Beckhoff EQ3xxx/Beckhoff EQ3xxxEK1122/A_0002(EQ3174-0002-0017)
//     PlcTask Inputs/GVL_iXlinker.EtherCAT_Master_EQxxxx.Beckhoff_EQ3xxx.Beckhoff_EQ3xxxEK1122.A_0002_EQ3174_0002_0017.AI_Standard_Channel_1.Status/Underrange <-> AI Standard Channel 1/Status/Underrange
//     PlcTask Inputs/GVL_iXlinker.EtherCAT_Master_EQxxxx.Beckhoff_EQ3xxx.Beckhoff_EQ3xxxEK1122.A_0002_EQ3174_0002_0017.AI_Standard_Channel_2.Status/Underrange <-> AI Standard Channel 2/Status/Underrange
//     PlcTask Inputs/GVL_iXlinker.EtherCAT_Master_EQxxxx.Beckhoff_EQ3xxx.Beckhoff_EQ3xxxEK1122.A_0002_EQ3174_0002_0017.AI_Standard_Channel_3.Status/Underrange <-> AI Standard Channel 3/Status/Underrange
//     PlcTask Inputs/GVL_iXlinker.EtherCAT_Master_EQxxxx.Beckhoff_EQ3xxx.Beckhoff_EQ3xxxEK1122.A_0002_EQ3174_0002_0017.AI_Standard_Channel_4.Status/Underrange <-> AI Standard Channel 4/Status/Underrange
//     PlcTask Inputs/GVL_iXlinker.EtherCAT_Master_EQxxxx.Beckhoff_EQ3xxx.Beckhoff_EQ3xxxEK1122.A_0002_EQ3174_0002_0017.AI_Standard_Channel_1.Status/Overrange <-> AI Standard Channel 1/Status/Overrange
//     PlcTask Inputs/GVL_iXlinker.EtherCAT_Master_EQxxxx.Beckhoff_EQ3xxx.Beckhoff_EQ3xxxEK1122.A_0002_EQ3174_0002_0017.AI_Standard_Channel_2.Status/Overrange <-> AI Standard Channel 2/Status/Overrange
//     PlcTask Inputs/GVL_iXlinker.EtherCAT_Master_EQxxxx.Beckhoff_EQ3xxx.Beckhoff_EQ3xxxEK1122.A_0002_EQ3174_0002_0017.AI_Standard_Channel_3.Status/Overrange <-> AI Standard Channel 3/Status/Overrange
//     PlcTask Inputs/GVL_iXlinker.EtherCAT_Master_EQxxxx.Beckhoff_EQ3xxx.Beckhoff_EQ3xxxEK1122.A_0002_EQ3174_0002_0017.AI_Standard_Channel_4.Status/Overrange <-> AI Standard Channel 4/Status/Overrange
//     PlcTask Inputs/GVL_iXlinker.EtherCAT_Master_EQxxxx.Beckhoff_EQ3xxx.Beckhoff_EQ3xxxEK1122.A_0002_EQ3174_0002_0017.AI_Standard_Channel_1.Status/Limit_1 <-> AI Standard Channel 1/Status/Limit 1
//     PlcTask Inputs/GVL_iXlinker.EtherCAT_Master_EQxxxx.Beckhoff_EQ3xxx.Beckhoff_EQ3xxxEK1122.A_0002_EQ3174_0002_0017.AI_Standard_Channel_1.Status/Limit_2 <-> AI Standard Channel 1/Status/Limit 2
//     PlcTask Inputs/GVL_iXlinker.EtherCAT_Master_EQxxxx.Beckhoff_EQ3xxx.Beckhoff_EQ3xxxEK1122.A_0002_EQ3174_0002_0017.AI_Standard_Channel_2.Status/Limit_1 <-> AI Standard Channel 2/Status/Limit 1
//     PlcTask Inputs/GVL_iXlinker.EtherCAT_Master_EQxxxx.Beckhoff_EQ3xxx.Beckhoff_EQ3xxxEK1122.A_0002_EQ3174_0002_0017.AI_Standard_Channel_2.Status/Limit_2 <-> AI Standard Channel 2/Status/Limit 2
//     PlcTask Inputs/GVL_iXlinker.EtherCAT_Master_EQxxxx.Beckhoff_EQ3xxx.Beckhoff_EQ3xxxEK1122.A_0002_EQ3174_0002_0017.AI_Standard_Channel_3.Status/Limit_1 <-> AI Standard Channel 3/Status/Limit 1
//     PlcTask Inputs/GVL_iXlinker.EtherCAT_Master_EQxxxx.Beckhoff_EQ3xxx.Beckhoff_EQ3xxxEK1122.A_0002_EQ3174_0002_0017.AI_Standard_Channel_3.Status/Limit_2 <-> AI Standard Channel 3/Status/Limit 2
//     PlcTask Inputs/GVL_iXlinker.EtherCAT_Master_EQxxxx.Beckhoff_EQ3xxx.Beckhoff_EQ3xxxEK1122.A_0002_EQ3174_0002_0017.AI_Standard_Channel_4.Status/Limit_1 <-> AI Standard Channel 4/Status/Limit 1
//     PlcTask Inputs/GVL_iXlinker.EtherCAT_Master_EQxxxx.Beckhoff_EQ3xxx.Beckhoff_EQ3xxxEK1122.A_0002_EQ3174_0002_0017.AI_Standard_Channel_4.Status/Limit_2 <-> AI Standard Channel 4/Status/Limit 2
//     PlcTask Inputs/GVL_iXlinker.EtherCAT_Master_EQxxxx.Beckhoff_EQ3xxx.Beckhoff_EQ3xxxEK1122.A_0002_EQ3174_0002_0017.AI_Standard_Channel_1.Status/Error <-> AI Standard Channel 1/Status/Error
//     PlcTask Inputs/GVL_iXlinker.EtherCAT_Master_EQxxxx.Beckhoff_EQ3xxx.Beckhoff_EQ3xxxEK1122.A_0002_EQ3174_0002_0017.AI_Standard_Channel_2.Status/Error <-> AI Standard Channel 2/Status/Error
//     PlcTask Inputs/GVL_iXlinker.EtherCAT_Master_EQxxxx.Beckhoff_EQ3xxx.Beckhoff_EQ3xxxEK1122.A_0002_EQ3174_0002_0017.AI_Standard_Channel_3.Status/Error <-> AI Standard Channel 3/Status/Error
//     PlcTask Inputs/GVL_iXlinker.EtherCAT_Master_EQxxxx.Beckhoff_EQ3xxx.Beckhoff_EQ3xxxEK1122.A_0002_EQ3174_0002_0017.AI_Standard_Channel_4.Status/Error <-> AI Standard Channel 4/Status/Error
//     PlcTask Inputs/GVL_iXlinker.EtherCAT_Master_EQxxxx.Beckhoff_EQ3xxx.Beckhoff_EQ3xxxEK1122.A_0002_EQ3174_0002_0017.AI_Standard_Channel_1.Status/Sync_error <-> AI Standard Channel 1/Status/Sync error
//     PlcTask Inputs/GVL_iXlinker.EtherCAT_Master_EQxxxx.Beckhoff_EQ3xxx.Beckhoff_EQ3xxxEK1122.A_0002_EQ3174_0002_0017.AI_Standard_Channel_2.Status/Sync_error <-> AI Standard Channel 2/Status/Sync error
//     PlcTask Inputs/GVL_iXlinker.EtherCAT_Master_EQxxxx.Beckhoff_EQ3xxx.Beckhoff_EQ3xxxEK1122.A_0002_EQ3174_0002_0017.AI_Standard_Channel_3.Status/Sync_error <-> AI Standard Channel 3/Status/Sync error
//     PlcTask Inputs/GVL_iXlinker.EtherCAT_Master_EQxxxx.Beckhoff_EQ3xxx.Beckhoff_EQ3xxxEK1122.A_0002_EQ3174_0002_0017.AI_Standard_Channel_4.Status/Sync_error <-> AI Standard Channel 4/Status/Sync error
//     PlcTask Inputs/GVL_iXlinker.EtherCAT_Master_EQxxxx.Beckhoff_EQ3xxx.Beckhoff_EQ3xxxEK1122.A_0002_EQ3174_0002_0017.AI_Standard_Channel_1.Status/TxPDO_State <-> AI Standard Channel 1/Status/TxPDO State
//     PlcTask Inputs/GVL_iXlinker.EtherCAT_Master_EQxxxx.Beckhoff_EQ3xxx.Beckhoff_EQ3xxxEK1122.A_0002_EQ3174_0002_0017.AI_Standard_Channel_2.Status/TxPDO_State <-> AI Standard Channel 2/Status/TxPDO State
//     PlcTask Inputs/GVL_iXlinker.EtherCAT_Master_EQxxxx.Beckhoff_EQ3xxx.Beckhoff_EQ3xxxEK1122.A_0002_EQ3174_0002_0017.AI_Standard_Channel_3.Status/TxPDO_State <-> AI Standard Channel 3/Status/TxPDO State
//     PlcTask Inputs/GVL_iXlinker.EtherCAT_Master_EQxxxx.Beckhoff_EQ3xxx.Beckhoff_EQ3xxxEK1122.A_0002_EQ3174_0002_0017.AI_Standard_Channel_4.Status/TxPDO_State <-> AI Standard Channel 4/Status/TxPDO State
//     PlcTask Inputs/GVL_iXlinker.EtherCAT_Master_EQxxxx.Beckhoff_EQ3xxx.Beckhoff_EQ3xxxEK1122.A_0002_EQ3174_0002_0017.AI_Standard_Channel_1.Status/TxPDO_Toggle <-> AI Standard Channel 1/Status/TxPDO Toggle
//     PlcTask Inputs/GVL_iXlinker.EtherCAT_Master_EQxxxx.Beckhoff_EQ3xxx.Beckhoff_EQ3xxxEK1122.A_0002_EQ3174_0002_0017.AI_Standard_Channel_2.Status/TxPDO_Toggle <-> AI Standard Channel 2/Status/TxPDO Toggle
//     PlcTask Inputs/GVL_iXlinker.EtherCAT_Master_EQxxxx.Beckhoff_EQ3xxx.Beckhoff_EQ3xxxEK1122.A_0002_EQ3174_0002_0017.AI_Standard_Channel_3.Status/TxPDO_Toggle <-> AI Standard Channel 3/Status/TxPDO Toggle
//     PlcTask Inputs/GVL_iXlinker.EtherCAT_Master_EQxxxx.Beckhoff_EQ3xxx.Beckhoff_EQ3xxxEK1122.A_0002_EQ3174_0002_0017.AI_Standard_Channel_4.Status/TxPDO_Toggle <-> AI Standard Channel 4/Status/TxPDO Toggle
//     PlcTask Inputs/GVL_iXlinker.EtherCAT_Master_EQxxxx.Beckhoff_EQ3xxx.Beckhoff_EQ3xxxEK1122.A_0002_EQ3174_0002_0017.AI_Standard_Channel_1.Value <-> AI Standard Channel 1/Value
//     PlcTask Inputs/GVL_iXlinker.EtherCAT_Master_EQxxxx.Beckhoff_EQ3xxx.Beckhoff_EQ3xxxEK1122.A_0002_EQ3174_0002_0017.AI_Standard_Channel_2.Value <-> AI Standard Channel 2/Value
//     PlcTask Inputs/GVL_iXlinker.EtherCAT_Master_EQxxxx.Beckhoff_EQ3xxx.Beckhoff_EQ3xxxEK1122.A_0002_EQ3174_0002_0017.AI_Standard_Channel_3.Value <-> AI Standard Channel 3/Value
//     PlcTask Inputs/GVL_iXlinker.EtherCAT_Master_EQxxxx.Beckhoff_EQ3xxx.Beckhoff_EQ3xxxEK1122.A_0002_EQ3174_0002_0017.AI_Standard_Channel_4.Value <-> AI Standard Channel 4/Value
//     PlcTask Inputs/GVL_iXlinker.EtherCAT_Master_EQxxxx.Beckhoff_EQ3xxx.Beckhoff_EQ3xxxEK1122.A_0002_EQ3174_0002_0017.WcState.WcState <-> WcState/WcState
//     PlcTask Inputs/GVL_iXlinker.EtherCAT_Master_EQxxxx.Beckhoff_EQ3xxx.Beckhoff_EQ3xxxEK1122.A_0002_EQ3174_0002_0017.WcState.InputToggle <-> WcState/InputToggle
//     PlcTask Inputs/GVL_iXlinker.EtherCAT_Master_EQxxxx.Beckhoff_EQ3xxx.Beckhoff_EQ3xxxEK1122.A_0002_EQ3174_0002_0017.InfoData.AdsAddr <-> InfoData/AdsAddr
//     PlcTask Inputs/GVL_iXlinker.EtherCAT_Master_EQxxxx.Beckhoff_EQ3xxx.Beckhoff_EQ3xxxEK1122.A_0002_EQ3174_0002_0017.InfoData.State <-> InfoData/State
//   PLC/PLC Instance <-> EtherCAT Master EQxxxx/Beckhoff EQ3xxx/Beckhoff EQ3xxxEK1122/A_0003(EQ3174-0002-0021)
//     PlcTask Inputs/GVL_iXlinker.EtherCAT_Master_EQxxxx.Beckhoff_EQ3xxx.Beckhoff_EQ3xxxEK1122.A_0003_EQ3174_0002_0021.AI_Standard_Channel_1.Status/Underrange <-> AI Standard Channel 1/Status/Underrange
//     PlcTask Inputs/GVL_iXlinker.EtherCAT_Master_EQxxxx.Beckhoff_EQ3xxx.Beckhoff_EQ3xxxEK1122.A_0003_EQ3174_0002_0021.AI_Standard_Channel_2.Status/Underrange <-> AI Standard Channel 2/Status/Underrange
//     PlcTask Inputs/GVL_iXlinker.EtherCAT_Master_EQxxxx.Beckhoff_EQ3xxx.Beckhoff_EQ3xxxEK1122.A_0003_EQ3174_0002_0021.AI_Standard_Channel_3.Status/Underrange <-> AI Standard Channel 3/Status/Underrange
//     PlcTask Inputs/GVL_iXlinker.EtherCAT_Master_EQxxxx.Beckhoff_EQ3xxx.Beckhoff_EQ3xxxEK1122.A_0003_EQ3174_0002_0021.AI_Standard_Channel_4.Status/Underrange <-> AI Standard Channel 4/Status/Underrange
//     PlcTask Inputs/GVL_iXlinker.EtherCAT_Master_EQxxxx.Beckhoff_EQ3xxx.Beckhoff_EQ3xxxEK1122.A_0003_EQ3174_0002_0021.AI_Standard_Channel_1.Status/Overrange <-> AI Standard Channel 1/Status/Overrange
//     PlcTask Inputs/GVL_iXlinker.EtherCAT_Master_EQxxxx.Beckhoff_EQ3xxx.Beckhoff_EQ3xxxEK1122.A_0003_EQ3174_0002_0021.AI_Standard_Channel_2.Status/Overrange <-> AI Standard Channel 2/Status/Overrange
//     PlcTask Inputs/GVL_iXlinker.EtherCAT_Master_EQxxxx.Beckhoff_EQ3xxx.Beckhoff_EQ3xxxEK1122.A_0003_EQ3174_0002_0021.AI_Standard_Channel_3.Status/Overrange <-> AI Standard Channel 3/Status/Overrange
//     PlcTask Inputs/GVL_iXlinker.EtherCAT_Master_EQxxxx.Beckhoff_EQ3xxx.Beckhoff_EQ3xxxEK1122.A_0003_EQ3174_0002_0021.AI_Standard_Channel_4.Status/Overrange <-> AI Standard Channel 4/Status/Overrange
//     PlcTask Inputs/GVL_iXlinker.EtherCAT_Master_EQxxxx.Beckhoff_EQ3xxx.Beckhoff_EQ3xxxEK1122.A_0003_EQ3174_0002_0021.AI_Standard_Channel_1.Status/Limit_1 <-> AI Standard Channel 1/Status/Limit 1
//     PlcTask Inputs/GVL_iXlinker.EtherCAT_Master_EQxxxx.Beckhoff_EQ3xxx.Beckhoff_EQ3xxxEK1122.A_0003_EQ3174_0002_0021.AI_Standard_Channel_1.Status/Limit_2 <-> AI Standard Channel 1/Status/Limit 2
//     PlcTask Inputs/GVL_iXlinker.EtherCAT_Master_EQxxxx.Beckhoff_EQ3xxx.Beckhoff_EQ3xxxEK1122.A_0003_EQ3174_0002_0021.AI_Standard_Channel_2.Status/Limit_1 <-> AI Standard Channel 2/Status/Limit 1
//     PlcTask Inputs/GVL_iXlinker.EtherCAT_Master_EQxxxx.Beckhoff_EQ3xxx.Beckhoff_EQ3xxxEK1122.A_0003_EQ3174_0002_0021.AI_Standard_Channel_2.Status/Limit_2 <-> AI Standard Channel 2/Status/Limit 2
//     PlcTask Inputs/GVL_iXlinker.EtherCAT_Master_EQxxxx.Beckhoff_EQ3xxx.Beckhoff_EQ3xxxEK1122.A_0003_EQ3174_0002_0021.AI_Standard_Channel_3.Status/Limit_1 <-> AI Standard Channel 3/Status/Limit 1
//     PlcTask Inputs/GVL_iXlinker.EtherCAT_Master_EQxxxx.Beckhoff_EQ3xxx.Beckhoff_EQ3xxxEK1122.A_0003_EQ3174_0002_0021.AI_Standard_Channel_3.Status/Limit_2 <-> AI Standard Channel 3/Status/Limit 2
//     PlcTask Inputs/GVL_iXlinker.EtherCAT_Master_EQxxxx.Beckhoff_EQ3xxx.Beckhoff_EQ3xxxEK1122.A_0003_EQ3174_0002_0021.AI_Standard_Channel_4.Status/Limit_1 <-> AI Standard Channel 4/Status/Limit 1
//     PlcTask Inputs/GVL_iXlinker.EtherCAT_Master_EQxxxx.Beckhoff_EQ3xxx.Beckhoff_EQ3xxxEK1122.A_0003_EQ3174_0002_0021.AI_Standard_Channel_4.Status/Limit_2 <-> AI Standard Channel 4/Status/Limit 2
//     PlcTask Inputs/GVL_iXlinker.EtherCAT_Master_EQxxxx.Beckhoff_EQ3xxx.Beckhoff_EQ3xxxEK1122.A_0003_EQ3174_0002_0021.AI_Standard_Channel_1.Status/Error <-> AI Standard Channel 1/Status/Error
//     PlcTask Inputs/GVL_iXlinker.EtherCAT_Master_EQxxxx.Beckhoff_EQ3xxx.Beckhoff_EQ3xxxEK1122.A_0003_EQ3174_0002_0021.AI_Standard_Channel_2.Status/Error <-> AI Standard Channel 2/Status/Error
//     PlcTask Inputs/GVL_iXlinker.EtherCAT_Master_EQxxxx.Beckhoff_EQ3xxx.Beckhoff_EQ3xxxEK1122.A_0003_EQ3174_0002_0021.AI_Standard_Channel_3.Status/Error <-> AI Standard Channel 3/Status/Error
//     PlcTask Inputs/GVL_iXlinker.EtherCAT_Master_EQxxxx.Beckhoff_EQ3xxx.Beckhoff_EQ3xxxEK1122.A_0003_EQ3174_0002_0021.AI_Standard_Channel_4.Status/Error <-> AI Standard Channel 4/Status/Error
//     PlcTask Inputs/GVL_iXlinker.EtherCAT_Master_EQxxxx.Beckhoff_EQ3xxx.Beckhoff_EQ3xxxEK1122.A_0003_EQ3174_0002_0021.AI_Standard_Channel_1.Status/Sync_error <-> AI Standard Channel 1/Status/Sync error
//     PlcTask Inputs/GVL_iXlinker.EtherCAT_Master_EQxxxx.Beckhoff_EQ3xxx.Beckhoff_EQ3xxxEK1122.A_0003_EQ3174_0002_0021.AI_Standard_Channel_2.Status/Sync_error <-> AI Standard Channel 2/Status/Sync error
//     PlcTask Inputs/GVL_iXlinker.EtherCAT_Master_EQxxxx.Beckhoff_EQ3xxx.Beckhoff_EQ3xxxEK1122.A_0003_EQ3174_0002_0021.AI_Standard_Channel_3.Status/Sync_error <-> AI Standard Channel 3/Status/Sync error
//     PlcTask Inputs/GVL_iXlinker.EtherCAT_Master_EQxxxx.Beckhoff_EQ3xxx.Beckhoff_EQ3xxxEK1122.A_0003_EQ3174_0002_0021.AI_Standard_Channel_4.Status/Sync_error <-> AI Standard Channel 4/Status/Sync error
//     PlcTask Inputs/GVL_iXlinker.EtherCAT_Master_EQxxxx.Beckhoff_EQ3xxx.Beckhoff_EQ3xxxEK1122.A_0003_EQ3174_0002_0021.AI_Standard_Channel_1.Status/TxPDO_State <-> AI Standard Channel 1/Status/TxPDO State
//     PlcTask Inputs/GVL_iXlinker.EtherCAT_Master_EQxxxx.Beckhoff_EQ3xxx.Beckhoff_EQ3xxxEK1122.A_0003_EQ3174_0002_0021.AI_Standard_Channel_2.Status/TxPDO_State <-> AI Standard Channel 2/Status/TxPDO State
//     PlcTask Inputs/GVL_iXlinker.EtherCAT_Master_EQxxxx.Beckhoff_EQ3xxx.Beckhoff_EQ3xxxEK1122.A_0003_EQ3174_0002_0021.AI_Standard_Channel_3.Status/TxPDO_State <-> AI Standard Channel 3/Status/TxPDO State
//     PlcTask Inputs/GVL_iXlinker.EtherCAT_Master_EQxxxx.Beckhoff_EQ3xxx.Beckhoff_EQ3xxxEK1122.A_0003_EQ3174_0002_0021.AI_Standard_Channel_4.Status/TxPDO_State <-> AI Standard Channel 4/Status/TxPDO State
//     PlcTask Inputs/GVL_iXlinker.EtherCAT_Master_EQxxxx.Beckhoff_EQ3xxx.Beckhoff_EQ3xxxEK1122.A_0003_EQ3174_0002_0021.AI_Standard_Channel_1.Status/TxPDO_Toggle <-> AI Standard Channel 1/Status/TxPDO Toggle
//     PlcTask Inputs/GVL_iXlinker.EtherCAT_Master_EQxxxx.Beckhoff_EQ3xxx.Beckhoff_EQ3xxxEK1122.A_0003_EQ3174_0002_0021.AI_Standard_Channel_2.Status/TxPDO_Toggle <-> AI Standard Channel 2/Status/TxPDO Toggle
//     PlcTask Inputs/GVL_iXlinker.EtherCAT_Master_EQxxxx.Beckhoff_EQ3xxx.Beckhoff_EQ3xxxEK1122.A_0003_EQ3174_0002_0021.AI_Standard_Channel_3.Status/TxPDO_Toggle <-> AI Standard Channel 3/Status/TxPDO Toggle
//     PlcTask Inputs/GVL_iXlinker.EtherCAT_Master_EQxxxx.Beckhoff_EQ3xxx.Beckhoff_EQ3xxxEK1122.A_0003_EQ3174_0002_0021.AI_Standard_Channel_4.Status/TxPDO_Toggle <-> AI Standard Channel 4/Status/TxPDO Toggle
//     PlcTask Inputs/GVL_iXlinker.EtherCAT_Master_EQxxxx.Beckhoff_EQ3xxx.Beckhoff_EQ3xxxEK1122.A_0003_EQ3174_0002_0021.AI_Standard_Channel_1.Value <-> AI Standard Channel 1/Value
//     PlcTask Inputs/GVL_iXlinker.EtherCAT_Master_EQxxxx.Beckhoff_EQ3xxx.Beckhoff_EQ3xxxEK1122.A_0003_EQ3174_0002_0021.AI_Standard_Channel_2.Value <-> AI Standard Channel 2/Value
//     PlcTask Inputs/GVL_iXlinker.EtherCAT_Master_EQxxxx.Beckhoff_EQ3xxx.Beckhoff_EQ3xxxEK1122.A_0003_EQ3174_0002_0021.AI_Standard_Channel_3.Value <-> AI Standard Channel 3/Value
//     PlcTask Inputs/GVL_iXlinker.EtherCAT_Master_EQxxxx.Beckhoff_EQ3xxx.Beckhoff_EQ3xxxEK1122.A_0003_EQ3174_0002_0021.AI_Standard_Channel_4.Value <-> AI Standard Channel 4/Value
//     PlcTask Inputs/GVL_iXlinker.EtherCAT_Master_EQxxxx.Beckhoff_EQ3xxx.Beckhoff_EQ3xxxEK1122.A_0003_EQ3174_0002_0021.WcState.WcState <-> WcState/WcState
//     PlcTask Inputs/GVL_iXlinker.EtherCAT_Master_EQxxxx.Beckhoff_EQ3xxx.Beckhoff_EQ3xxxEK1122.A_0003_EQ3174_0002_0021.WcState.InputToggle <-> WcState/InputToggle
//     PlcTask Inputs/GVL_iXlinker.EtherCAT_Master_EQxxxx.Beckhoff_EQ3xxx.Beckhoff_EQ3xxxEK1122.A_0003_EQ3174_0002_0021.InfoData.AdsAddr <-> InfoData/AdsAddr
//     PlcTask Inputs/GVL_iXlinker.EtherCAT_Master_EQxxxx.Beckhoff_EQ3xxx.Beckhoff_EQ3xxxEK1122.A_0003_EQ3174_0002_0021.InfoData.State <-> InfoData/State
//   PLC/PLC Instance <-> EtherCAT Master EQxxxx/Beckhoff EQ3xxx/Beckhoff EQ3xxxEK1122/A_0004(EQ3174-0002-0022)
//     PlcTask Inputs/GVL_iXlinker.EtherCAT_Master_EQxxxx.Beckhoff_EQ3xxx.Beckhoff_EQ3xxxEK1122.A_0004_EQ3174_0002_0022.AI_Standard_Channel_1.Status/Underrange <-> AI Standard Channel 1/Status/Underrange
//     PlcTask Inputs/GVL_iXlinker.EtherCAT_Master_EQxxxx.Beckhoff_EQ3xxx.Beckhoff_EQ3xxxEK1122.A_0004_EQ3174_0002_0022.AI_Standard_Channel_2.Status/Underrange <-> AI Standard Channel 2/Status/Underrange
//     PlcTask Inputs/GVL_iXlinker.EtherCAT_Master_EQxxxx.Beckhoff_EQ3xxx.Beckhoff_EQ3xxxEK1122.A_0004_EQ3174_0002_0022.AI_Standard_Channel_3.Status/Underrange <-> AI Standard Channel 3/Status/Underrange
//     PlcTask Inputs/GVL_iXlinker.EtherCAT_Master_EQxxxx.Beckhoff_EQ3xxx.Beckhoff_EQ3xxxEK1122.A_0004_EQ3174_0002_0022.AI_Standard_Channel_4.Status/Underrange <-> AI Standard Channel 4/Status/Underrange
//     PlcTask Inputs/GVL_iXlinker.EtherCAT_Master_EQxxxx.Beckhoff_EQ3xxx.Beckhoff_EQ3xxxEK1122.A_0004_EQ3174_0002_0022.AI_Standard_Channel_1.Status/Overrange <-> AI Standard Channel 1/Status/Overrange
//     PlcTask Inputs/GVL_iXlinker.EtherCAT_Master_EQxxxx.Beckhoff_EQ3xxx.Beckhoff_EQ3xxxEK1122.A_0004_EQ3174_0002_0022.AI_Standard_Channel_2.Status/Overrange <-> AI Standard Channel 2/Status/Overrange
//     PlcTask Inputs/GVL_iXlinker.EtherCAT_Master_EQxxxx.Beckhoff_EQ3xxx.Beckhoff_EQ3xxxEK1122.A_0004_EQ3174_0002_0022.AI_Standard_Channel_3.Status/Overrange <-> AI Standard Channel 3/Status/Overrange
//     PlcTask Inputs/GVL_iXlinker.EtherCAT_Master_EQxxxx.Beckhoff_EQ3xxx.Beckhoff_EQ3xxxEK1122.A_0004_EQ3174_0002_0022.AI_Standard_Channel_4.Status/Overrange <-> AI Standard Channel 4/Status/Overrange
//     PlcTask Inputs/GVL_iXlinker.EtherCAT_Master_EQxxxx.Beckhoff_EQ3xxx.Beckhoff_EQ3xxxEK1122.A_0004_EQ3174_0002_0022.AI_Standard_Channel_1.Status/Limit_1 <-> AI Standard Channel 1/Status/Limit 1
//     PlcTask Inputs/GVL_iXlinker.EtherCAT_Master_EQxxxx.Beckhoff_EQ3xxx.Beckhoff_EQ3xxxEK1122.A_0004_EQ3174_0002_0022.AI_Standard_Channel_1.Status/Limit_2 <-> AI Standard Channel 1/Status/Limit 2
//     PlcTask Inputs/GVL_iXlinker.EtherCAT_Master_EQxxxx.Beckhoff_EQ3xxx.Beckhoff_EQ3xxxEK1122.A_0004_EQ3174_0002_0022.AI_Standard_Channel_2.Status/Limit_1 <-> AI Standard Channel 2/Status/Limit 1
//     PlcTask Inputs/GVL_iXlinker.EtherCAT_Master_EQxxxx.Beckhoff_EQ3xxx.Beckhoff_EQ3xxxEK1122.A_0004_EQ3174_0002_0022.AI_Standard_Channel_2.Status/Limit_2 <-> AI Standard Channel 2/Status/Limit 2
//     PlcTask Inputs/GVL_iXlinker.EtherCAT_Master_EQxxxx.Beckhoff_EQ3xxx.Beckhoff_EQ3xxxEK1122.A_0004_EQ3174_0002_0022.AI_Standard_Channel_3.Status/Limit_1 <-> AI Standard Channel 3/Status/Limit 1
//     PlcTask Inputs/GVL_iXlinker.EtherCAT_Master_EQxxxx.Beckhoff_EQ3xxx.Beckhoff_EQ3xxxEK1122.A_0004_EQ3174_0002_0022.AI_Standard_Channel_3.Status/Limit_2 <-> AI Standard Channel 3/Status/Limit 2
//     PlcTask Inputs/GVL_iXlinker.EtherCAT_Master_EQxxxx.Beckhoff_EQ3xxx.Beckhoff_EQ3xxxEK1122.A_0004_EQ3174_0002_0022.AI_Standard_Channel_4.Status/Limit_1 <-> AI Standard Channel 4/Status/Limit 1
//     PlcTask Inputs/GVL_iXlinker.EtherCAT_Master_EQxxxx.Beckhoff_EQ3xxx.Beckhoff_EQ3xxxEK1122.A_0004_EQ3174_0002_0022.AI_Standard_Channel_4.Status/Limit_2 <-> AI Standard Channel 4/Status/Limit 2
//     PlcTask Inputs/GVL_iXlinker.EtherCAT_Master_EQxxxx.Beckhoff_EQ3xxx.Beckhoff_EQ3xxxEK1122.A_0004_EQ3174_0002_0022.AI_Standard_Channel_1.Status/Error <-> AI Standard Channel 1/Status/Error
//     PlcTask Inputs/GVL_iXlinker.EtherCAT_Master_EQxxxx.Beckhoff_EQ3xxx.Beckhoff_EQ3xxxEK1122.A_0004_EQ3174_0002_0022.AI_Standard_Channel_2.Status/Error <-> AI Standard Channel 2/Status/Error
//     PlcTask Inputs/GVL_iXlinker.EtherCAT_Master_EQxxxx.Beckhoff_EQ3xxx.Beckhoff_EQ3xxxEK1122.A_0004_EQ3174_0002_0022.AI_Standard_Channel_3.Status/Error <-> AI Standard Channel 3/Status/Error
//     PlcTask Inputs/GVL_iXlinker.EtherCAT_Master_EQxxxx.Beckhoff_EQ3xxx.Beckhoff_EQ3xxxEK1122.A_0004_EQ3174_0002_0022.AI_Standard_Channel_4.Status/Error <-> AI Standard Channel 4/Status/Error
//     PlcTask Inputs/GVL_iXlinker.EtherCAT_Master_EQxxxx.Beckhoff_EQ3xxx.Beckhoff_EQ3xxxEK1122.A_0004_EQ3174_0002_0022.AI_Standard_Channel_1.Status/Sync_error <-> AI Standard Channel 1/Status/Sync error
//     PlcTask Inputs/GVL_iXlinker.EtherCAT_Master_EQxxxx.Beckhoff_EQ3xxx.Beckhoff_EQ3xxxEK1122.A_0004_EQ3174_0002_0022.AI_Standard_Channel_2.Status/Sync_error <-> AI Standard Channel 2/Status/Sync error
//     PlcTask Inputs/GVL_iXlinker.EtherCAT_Master_EQxxxx.Beckhoff_EQ3xxx.Beckhoff_EQ3xxxEK1122.A_0004_EQ3174_0002_0022.AI_Standard_Channel_3.Status/Sync_error <-> AI Standard Channel 3/Status/Sync error
//     PlcTask Inputs/GVL_iXlinker.EtherCAT_Master_EQxxxx.Beckhoff_EQ3xxx.Beckhoff_EQ3xxxEK1122.A_0004_EQ3174_0002_0022.AI_Standard_Channel_4.Status/Sync_error <-> AI Standard Channel 4/Status/Sync error
//     PlcTask Inputs/GVL_iXlinker.EtherCAT_Master_EQxxxx.Beckhoff_EQ3xxx.Beckhoff_EQ3xxxEK1122.A_0004_EQ3174_0002_0022.AI_Standard_Channel_1.Status/TxPDO_State <-> AI Standard Channel 1/Status/TxPDO State
//     PlcTask Inputs/GVL_iXlinker.EtherCAT_Master_EQxxxx.Beckhoff_EQ3xxx.Beckhoff_EQ3xxxEK1122.A_0004_EQ3174_0002_0022.AI_Standard_Channel_2.Status/TxPDO_State <-> AI Standard Channel 2/Status/TxPDO State
//     PlcTask Inputs/GVL_iXlinker.EtherCAT_Master_EQxxxx.Beckhoff_EQ3xxx.Beckhoff_EQ3xxxEK1122.A_0004_EQ3174_0002_0022.AI_Standard_Channel_3.Status/TxPDO_State <-> AI Standard Channel 3/Status/TxPDO State
//     PlcTask Inputs/GVL_iXlinker.EtherCAT_Master_EQxxxx.Beckhoff_EQ3xxx.Beckhoff_EQ3xxxEK1122.A_0004_EQ3174_0002_0022.AI_Standard_Channel_4.Status/TxPDO_State <-> AI Standard Channel 4/Status/TxPDO State
//     PlcTask Inputs/GVL_iXlinker.EtherCAT_Master_EQxxxx.Beckhoff_EQ3xxx.Beckhoff_EQ3xxxEK1122.A_0004_EQ3174_0002_0022.AI_Standard_Channel_1.Status/TxPDO_Toggle <-> AI Standard Channel 1/Status/TxPDO Toggle
//     PlcTask Inputs/GVL_iXlinker.EtherCAT_Master_EQxxxx.Beckhoff_EQ3xxx.Beckhoff_EQ3xxxEK1122.A_0004_EQ3174_0002_0022.AI_Standard_Channel_2.Status/TxPDO_Toggle <-> AI Standard Channel 2/Status/TxPDO Toggle
//     PlcTask Inputs/GVL_iXlinker.EtherCAT_Master_EQxxxx.Beckhoff_EQ3xxx.Beckhoff_EQ3xxxEK1122.A_0004_EQ3174_0002_0022.AI_Standard_Channel_3.Status/TxPDO_Toggle <-> AI Standard Channel 3/Status/TxPDO Toggle
//     PlcTask Inputs/GVL_iXlinker.EtherCAT_Master_EQxxxx.Beckhoff_EQ3xxx.Beckhoff_EQ3xxxEK1122.A_0004_EQ3174_0002_0022.AI_Standard_Channel_4.Status/TxPDO_Toggle <-> AI Standard Channel 4/Status/TxPDO Toggle
//     PlcTask Inputs/GVL_iXlinker.EtherCAT_Master_EQxxxx.Beckhoff_EQ3xxx.Beckhoff_EQ3xxxEK1122.A_0004_EQ3174_0002_0022.AI_Standard_Channel_1.Value <-> AI Standard Channel 1/Value
//     PlcTask Inputs/GVL_iXlinker.EtherCAT_Master_EQxxxx.Beckhoff_EQ3xxx.Beckhoff_EQ3xxxEK1122.A_0004_EQ3174_0002_0022.AI_Standard_Channel_2.Value <-> AI Standard Channel 2/Value
//     PlcTask Inputs/GVL_iXlinker.EtherCAT_Master_EQxxxx.Beckhoff_EQ3xxx.Beckhoff_EQ3xxxEK1122.A_0004_EQ3174_0002_0022.AI_Standard_Channel_3.Value <-> AI Standard Channel 3/Value
//     PlcTask Inputs/GVL_iXlinker.EtherCAT_Master_EQxxxx.Beckhoff_EQ3xxx.Beckhoff_EQ3xxxEK1122.A_0004_EQ3174_0002_0022.AI_Standard_Channel_4.Value <-> AI Standard Channel 4/Value
//     PlcTask Inputs/GVL_iXlinker.EtherCAT_Master_EQxxxx.Beckhoff_EQ3xxx.Beckhoff_EQ3xxxEK1122.A_0004_EQ3174_0002_0022.WcState.WcState <-> WcState/WcState
//     PlcTask Inputs/GVL_iXlinker.EtherCAT_Master_EQxxxx.Beckhoff_EQ3xxx.Beckhoff_EQ3xxxEK1122.A_0004_EQ3174_0002_0022.WcState.InputToggle <-> WcState/InputToggle
//     PlcTask Inputs/GVL_iXlinker.EtherCAT_Master_EQxxxx.Beckhoff_EQ3xxx.Beckhoff_EQ3xxxEK1122.A_0004_EQ3174_0002_0022.InfoData.AdsAddr <-> InfoData/AdsAddr
//     PlcTask Inputs/GVL_iXlinker.EtherCAT_Master_EQxxxx.Beckhoff_EQ3xxx.Beckhoff_EQ3xxxEK1122.A_0004_EQ3174_0002_0022.InfoData.State <-> InfoData/State
//   PLC/PLC Instance <-> EtherCAT Master EQxxxx/Beckhoff EQ3xxx/Beckhoff EQ3xxxEK1122/A_0005(EQ3174-0002-0023)
//     PlcTask Inputs/GVL_iXlinker.EtherCAT_Master_EQxxxx.Beckhoff_EQ3xxx.Beckhoff_EQ3xxxEK1122.A_0005_EQ3174_0002_0023.AI_Standard_Channel_1.Status/Underrange <-> AI Standard Channel 1/Status/Underrange
//     PlcTask Inputs/GVL_iXlinker.EtherCAT_Master_EQxxxx.Beckhoff_EQ3xxx.Beckhoff_EQ3xxxEK1122.A_0005_EQ3174_0002_0023.AI_Standard_Channel_2.Status/Underrange <-> AI Standard Channel 2/Status/Underrange
//     PlcTask Inputs/GVL_iXlinker.EtherCAT_Master_EQxxxx.Beckhoff_EQ3xxx.Beckhoff_EQ3xxxEK1122.A_0005_EQ3174_0002_0023.AI_Standard_Channel_3.Status/Underrange <-> AI Standard Channel 3/Status/Underrange
//     PlcTask Inputs/GVL_iXlinker.EtherCAT_Master_EQxxxx.Beckhoff_EQ3xxx.Beckhoff_EQ3xxxEK1122.A_0005_EQ3174_0002_0023.AI_Standard_Channel_4.Status/Underrange <-> AI Standard Channel 4/Status/Underrange
//     PlcTask Inputs/GVL_iXlinker.EtherCAT_Master_EQxxxx.Beckhoff_EQ3xxx.Beckhoff_EQ3xxxEK1122.A_0005_EQ3174_0002_0023.AI_Standard_Channel_1.Status/Overrange <-> AI Standard Channel 1/Status/Overrange
//     PlcTask Inputs/GVL_iXlinker.EtherCAT_Master_EQxxxx.Beckhoff_EQ3xxx.Beckhoff_EQ3xxxEK1122.A_0005_EQ3174_0002_0023.AI_Standard_Channel_2.Status/Overrange <-> AI Standard Channel 2/Status/Overrange
//     PlcTask Inputs/GVL_iXlinker.EtherCAT_Master_EQxxxx.Beckhoff_EQ3xxx.Beckhoff_EQ3xxxEK1122.A_0005_EQ3174_0002_0023.AI_Standard_Channel_3.Status/Overrange <-> AI Standard Channel 3/Status/Overrange
//     PlcTask Inputs/GVL_iXlinker.EtherCAT_Master_EQxxxx.Beckhoff_EQ3xxx.Beckhoff_EQ3xxxEK1122.A_0005_EQ3174_0002_0023.AI_Standard_Channel_4.Status/Overrange <-> AI Standard Channel 4/Status/Overrange
//     PlcTask Inputs/GVL_iXlinker.EtherCAT_Master_EQxxxx.Beckhoff_EQ3xxx.Beckhoff_EQ3xxxEK1122.A_0005_EQ3174_0002_0023.AI_Standard_Channel_1.Status/Limit_1 <-> AI Standard Channel 1/Status/Limit 1
//     PlcTask Inputs/GVL_iXlinker.EtherCAT_Master_EQxxxx.Beckhoff_EQ3xxx.Beckhoff_EQ3xxxEK1122.A_0005_EQ3174_0002_0023.AI_Standard_Channel_1.Status/Limit_2 <-> AI Standard Channel 1/Status/Limit 2
//     PlcTask Inputs/GVL_iXlinker.EtherCAT_Master_EQxxxx.Beckhoff_EQ3xxx.Beckhoff_EQ3xxxEK1122.A_0005_EQ3174_0002_0023.AI_Standard_Channel_2.Status/Limit_1 <-> AI Standard Channel 2/Status/Limit 1
//     PlcTask Inputs/GVL_iXlinker.EtherCAT_Master_EQxxxx.Beckhoff_EQ3xxx.Beckhoff_EQ3xxxEK1122.A_0005_EQ3174_0002_0023.AI_Standard_Channel_2.Status/Limit_2 <-> AI Standard Channel 2/Status/Limit 2
//     PlcTask Inputs/GVL_iXlinker.EtherCAT_Master_EQxxxx.Beckhoff_EQ3xxx.Beckhoff_EQ3xxxEK1122.A_0005_EQ3174_0002_0023.AI_Standard_Channel_3.Status/Limit_1 <-> AI Standard Channel 3/Status/Limit 1
//     PlcTask Inputs/GVL_iXlinker.EtherCAT_Master_EQxxxx.Beckhoff_EQ3xxx.Beckhoff_EQ3xxxEK1122.A_0005_EQ3174_0002_0023.AI_Standard_Channel_3.Status/Limit_2 <-> AI Standard Channel 3/Status/Limit 2
//     PlcTask Inputs/GVL_iXlinker.EtherCAT_Master_EQxxxx.Beckhoff_EQ3xxx.Beckhoff_EQ3xxxEK1122.A_0005_EQ3174_0002_0023.AI_Standard_Channel_4.Status/Limit_1 <-> AI Standard Channel 4/Status/Limit 1
//     PlcTask Inputs/GVL_iXlinker.EtherCAT_Master_EQxxxx.Beckhoff_EQ3xxx.Beckhoff_EQ3xxxEK1122.A_0005_EQ3174_0002_0023.AI_Standard_Channel_4.Status/Limit_2 <-> AI Standard Channel 4/Status/Limit 2
//     PlcTask Inputs/GVL_iXlinker.EtherCAT_Master_EQxxxx.Beckhoff_EQ3xxx.Beckhoff_EQ3xxxEK1122.A_0005_EQ3174_0002_0023.AI_Standard_Channel_1.Status/Error <-> AI Standard Channel 1/Status/Error
//     PlcTask Inputs/GVL_iXlinker.EtherCAT_Master_EQxxxx.Beckhoff_EQ3xxx.Beckhoff_EQ3xxxEK1122.A_0005_EQ3174_0002_0023.AI_Standard_Channel_2.Status/Error <-> AI Standard Channel 2/Status/Error
//     PlcTask Inputs/GVL_iXlinker.EtherCAT_Master_EQxxxx.Beckhoff_EQ3xxx.Beckhoff_EQ3xxxEK1122.A_0005_EQ3174_0002_0023.AI_Standard_Channel_3.Status/Error <-> AI Standard Channel 3/Status/Error
//     PlcTask Inputs/GVL_iXlinker.EtherCAT_Master_EQxxxx.Beckhoff_EQ3xxx.Beckhoff_EQ3xxxEK1122.A_0005_EQ3174_0002_0023.AI_Standard_Channel_4.Status/Error <-> AI Standard Channel 4/Status/Error
//     PlcTask Inputs/GVL_iXlinker.EtherCAT_Master_EQxxxx.Beckhoff_EQ3xxx.Beckhoff_EQ3xxxEK1122.A_0005_EQ3174_0002_0023.AI_Standard_Channel_1.Status/Sync_error <-> AI Standard Channel 1/Status/Sync error
//     PlcTask Inputs/GVL_iXlinker.EtherCAT_Master_EQxxxx.Beckhoff_EQ3xxx.Beckhoff_EQ3xxxEK1122.A_0005_EQ3174_0002_0023.AI_Standard_Channel_2.Status/Sync_error <-> AI Standard Channel 2/Status/Sync error
//     PlcTask Inputs/GVL_iXlinker.EtherCAT_Master_EQxxxx.Beckhoff_EQ3xxx.Beckhoff_EQ3xxxEK1122.A_0005_EQ3174_0002_0023.AI_Standard_Channel_3.Status/Sync_error <-> AI Standard Channel 3/Status/Sync error
//     PlcTask Inputs/GVL_iXlinker.EtherCAT_Master_EQxxxx.Beckhoff_EQ3xxx.Beckhoff_EQ3xxxEK1122.A_0005_EQ3174_0002_0023.AI_Standard_Channel_4.Status/Sync_error <-> AI Standard Channel 4/Status/Sync error
//     PlcTask Inputs/GVL_iXlinker.EtherCAT_Master_EQxxxx.Beckhoff_EQ3xxx.Beckhoff_EQ3xxxEK1122.A_0005_EQ3174_0002_0023.AI_Standard_Channel_1.Status/TxPDO_State <-> AI Standard Channel 1/Status/TxPDO State
//     PlcTask Inputs/GVL_iXlinker.EtherCAT_Master_EQxxxx.Beckhoff_EQ3xxx.Beckhoff_EQ3xxxEK1122.A_0005_EQ3174_0002_0023.AI_Standard_Channel_2.Status/TxPDO_State <-> AI Standard Channel 2/Status/TxPDO State
//     PlcTask Inputs/GVL_iXlinker.EtherCAT_Master_EQxxxx.Beckhoff_EQ3xxx.Beckhoff_EQ3xxxEK1122.A_0005_EQ3174_0002_0023.AI_Standard_Channel_3.Status/TxPDO_State <-> AI Standard Channel 3/Status/TxPDO State
//     PlcTask Inputs/GVL_iXlinker.EtherCAT_Master_EQxxxx.Beckhoff_EQ3xxx.Beckhoff_EQ3xxxEK1122.A_0005_EQ3174_0002_0023.AI_Standard_Channel_4.Status/TxPDO_State <-> AI Standard Channel 4/Status/TxPDO State
//     PlcTask Inputs/GVL_iXlinker.EtherCAT_Master_EQxxxx.Beckhoff_EQ3xxx.Beckhoff_EQ3xxxEK1122.A_0005_EQ3174_0002_0023.AI_Standard_Channel_1.Status/TxPDO_Toggle <-> AI Standard Channel 1/Status/TxPDO Toggle
//     PlcTask Inputs/GVL_iXlinker.EtherCAT_Master_EQxxxx.Beckhoff_EQ3xxx.Beckhoff_EQ3xxxEK1122.A_0005_EQ3174_0002_0023.AI_Standard_Channel_2.Status/TxPDO_Toggle <-> AI Standard Channel 2/Status/TxPDO Toggle
//     PlcTask Inputs/GVL_iXlinker.EtherCAT_Master_EQxxxx.Beckhoff_EQ3xxx.Beckhoff_EQ3xxxEK1122.A_0005_EQ3174_0002_0023.AI_Standard_Channel_3.Status/TxPDO_Toggle <-> AI Standard Channel 3/Status/TxPDO Toggle
//     PlcTask Inputs/GVL_iXlinker.EtherCAT_Master_EQxxxx.Beckhoff_EQ3xxx.Beckhoff_EQ3xxxEK1122.A_0005_EQ3174_0002_0023.AI_Standard_Channel_4.Status/TxPDO_Toggle <-> AI Standard Channel 4/Status/TxPDO Toggle
//     PlcTask Inputs/GVL_iXlinker.EtherCAT_Master_EQxxxx.Beckhoff_EQ3xxx.Beckhoff_EQ3xxxEK1122.A_0005_EQ3174_0002_0023.AI_Standard_Channel_1.Value <-> AI Standard Channel 1/Value
//     PlcTask Inputs/GVL_iXlinker.EtherCAT_Master_EQxxxx.Beckhoff_EQ3xxx.Beckhoff_EQ3xxxEK1122.A_0005_EQ3174_0002_0023.AI_Standard_Channel_2.Value <-> AI Standard Channel 2/Value
//     PlcTask Inputs/GVL_iXlinker.EtherCAT_Master_EQxxxx.Beckhoff_EQ3xxx.Beckhoff_EQ3xxxEK1122.A_0005_EQ3174_0002_0023.AI_Standard_Channel_3.Value <-> AI Standard Channel 3/Value
//     PlcTask Inputs/GVL_iXlinker.EtherCAT_Master_EQxxxx.Beckhoff_EQ3xxx.Beckhoff_EQ3xxxEK1122.A_0005_EQ3174_0002_0023.AI_Standard_Channel_4.Value <-> AI Standard Channel 4/Value
//     PlcTask Inputs/GVL_iXlinker.EtherCAT_Master_EQxxxx.Beckhoff_EQ3xxx.Beckhoff_EQ3xxxEK1122.A_0005_EQ3174_0002_0023.WcState.WcState <-> WcState/WcState
//     PlcTask Inputs/GVL_iXlinker.EtherCAT_Master_EQxxxx.Beckhoff_EQ3xxx.Beckhoff_EQ3xxxEK1122.A_0005_EQ3174_0002_0023.WcState.InputToggle <-> WcState/InputToggle
//     PlcTask Inputs/GVL_iXlinker.EtherCAT_Master_EQxxxx.Beckhoff_EQ3xxx.Beckhoff_EQ3xxxEK1122.A_0005_EQ3174_0002_0023.InfoData.AdsAddr <-> InfoData/AdsAddr
//     PlcTask Inputs/GVL_iXlinker.EtherCAT_Master_EQxxxx.Beckhoff_EQ3xxx.Beckhoff_EQ3xxxEK1122.A_0005_EQ3174_0002_0023.InfoData.State <-> InfoData/State
//   PLC/PLC Instance <-> EtherCAT Master EQxxxx/Beckhoff EQ3xxx/Beckhoff EQ3xxxEK1122/A_0006(EQ3204-0002-0016)
//     PlcTask Inputs/GVL_iXlinker.EtherCAT_Master_EQxxxx.Beckhoff_EQ3xxx.Beckhoff_EQ3xxxEK1122.A_0006_EQ3204_0002_0016.RTD_RTDInputs_Channel_1.Status/Underrange <-> RTD RTDInputs Channel 1/Status/Underrange
//     PlcTask Inputs/GVL_iXlinker.EtherCAT_Master_EQxxxx.Beckhoff_EQ3xxx.Beckhoff_EQ3xxxEK1122.A_0006_EQ3204_0002_0016.RTD_RTDInputs_Channel_2.Status/Underrange <-> RTD RTDInputs Channel 2/Status/Underrange
//     PlcTask Inputs/GVL_iXlinker.EtherCAT_Master_EQxxxx.Beckhoff_EQ3xxx.Beckhoff_EQ3xxxEK1122.A_0006_EQ3204_0002_0016.RTD_RTDInputs_Channel_3.Status/Underrange <-> RTD RTDInputs Channel 3/Status/Underrange
//     PlcTask Inputs/GVL_iXlinker.EtherCAT_Master_EQxxxx.Beckhoff_EQ3xxx.Beckhoff_EQ3xxxEK1122.A_0006_EQ3204_0002_0016.RTD_RTDInputs_Channel_4.Status/Underrange <-> RTD RTDInputs Channel 4/Status/Underrange
//     PlcTask Inputs/GVL_iXlinker.EtherCAT_Master_EQxxxx.Beckhoff_EQ3xxx.Beckhoff_EQ3xxxEK1122.A_0006_EQ3204_0002_0016.RTD_RTDInputs_Channel_1.Status/Overrange <-> RTD RTDInputs Channel 1/Status/Overrange
//     PlcTask Inputs/GVL_iXlinker.EtherCAT_Master_EQxxxx.Beckhoff_EQ3xxx.Beckhoff_EQ3xxxEK1122.A_0006_EQ3204_0002_0016.RTD_RTDInputs_Channel_2.Status/Overrange <-> RTD RTDInputs Channel 2/Status/Overrange
//     PlcTask Inputs/GVL_iXlinker.EtherCAT_Master_EQxxxx.Beckhoff_EQ3xxx.Beckhoff_EQ3xxxEK1122.A_0006_EQ3204_0002_0016.RTD_RTDInputs_Channel_3.Status/Overrange <-> RTD RTDInputs Channel 3/Status/Overrange
//     PlcTask Inputs/GVL_iXlinker.EtherCAT_Master_EQxxxx.Beckhoff_EQ3xxx.Beckhoff_EQ3xxxEK1122.A_0006_EQ3204_0002_0016.RTD_RTDInputs_Channel_4.Status/Overrange <-> RTD RTDInputs Channel 4/Status/Overrange
//     PlcTask Inputs/GVL_iXlinker.EtherCAT_Master_EQxxxx.Beckhoff_EQ3xxx.Beckhoff_EQ3xxxEK1122.A_0006_EQ3204_0002_0016.RTD_RTDInputs_Channel_1.Status/Limit_1 <-> RTD RTDInputs Channel 1/Status/Limit 1
//     PlcTask Inputs/GVL_iXlinker.EtherCAT_Master_EQxxxx.Beckhoff_EQ3xxx.Beckhoff_EQ3xxxEK1122.A_0006_EQ3204_0002_0016.RTD_RTDInputs_Channel_1.Status/Limit_2 <-> RTD RTDInputs Channel 1/Status/Limit 2
//     PlcTask Inputs/GVL_iXlinker.EtherCAT_Master_EQxxxx.Beckhoff_EQ3xxx.Beckhoff_EQ3xxxEK1122.A_0006_EQ3204_0002_0016.RTD_RTDInputs_Channel_2.Status/Limit_1 <-> RTD RTDInputs Channel 2/Status/Limit 1
//     PlcTask Inputs/GVL_iXlinker.EtherCAT_Master_EQxxxx.Beckhoff_EQ3xxx.Beckhoff_EQ3xxxEK1122.A_0006_EQ3204_0002_0016.RTD_RTDInputs_Channel_2.Status/Limit_2 <-> RTD RTDInputs Channel 2/Status/Limit 2
//     PlcTask Inputs/GVL_iXlinker.EtherCAT_Master_EQxxxx.Beckhoff_EQ3xxx.Beckhoff_EQ3xxxEK1122.A_0006_EQ3204_0002_0016.RTD_RTDInputs_Channel_3.Status/Limit_1 <-> RTD RTDInputs Channel 3/Status/Limit 1
//     PlcTask Inputs/GVL_iXlinker.EtherCAT_Master_EQxxxx.Beckhoff_EQ3xxx.Beckhoff_EQ3xxxEK1122.A_0006_EQ3204_0002_0016.RTD_RTDInputs_Channel_3.Status/Limit_2 <-> RTD RTDInputs Channel 3/Status/Limit 2
//     PlcTask Inputs/GVL_iXlinker.EtherCAT_Master_EQxxxx.Beckhoff_EQ3xxx.Beckhoff_EQ3xxxEK1122.A_0006_EQ3204_0002_0016.RTD_RTDInputs_Channel_4.Status/Limit_1 <-> RTD RTDInputs Channel 4/Status/Limit 1
